KUKA KRL program: EPS_2_25252_PD2_A_20250919023702.src

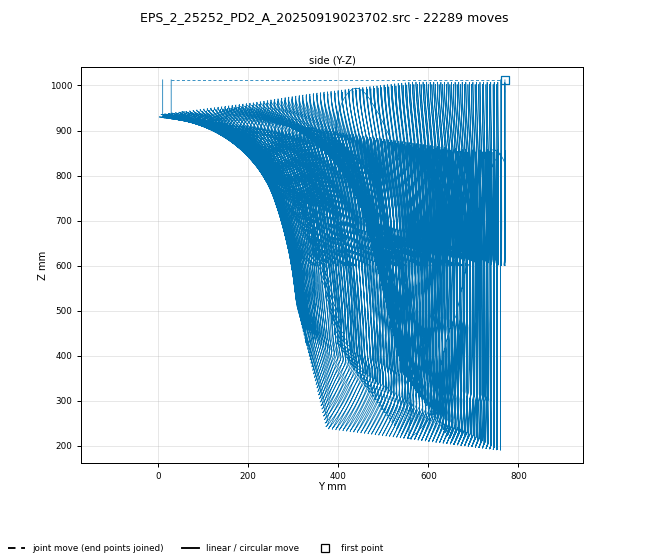
[picture p0: tool path of EPS_2_25252_PD2_A_20250919023702.src, 22289 of 22291 moves have a stored position in this frame; points joined in program order, loops and branches not executed]
&ACCESS RVP
&REL 4
&COMMENT QRS 19112012
&PARAM EDITMASK = *
DEF PART()
EXT BAS (BAS_COMMAND :IN,REAL :IN )
INT I
BAS (#INITMOV,0 )

;KUKA QRS Post kuka4.cps  Date:22-06-2017 !

File_ID=2839

QRS_PRE_INIT()

;Init var - Until changes are made in qrs_pre_init
Outlet_Square_prg=0
Inlet_1_Square_prg=0
Inlet_2_Square_prg=0
Inlet_3_Square_prg=0
Inlet_4_Square_prg=0
Inlet_5_Square_prg=0

Outlet_1={X 0.000, Y 562.000, Z 659.500, B 0.000, E1 0.000 }
Outlet_1={X 0.000, Y 562.000, Z 659.500, B 0.000, E1 0.000 }
Inlet_1={X 0.000, Y 675.710, Z 469.500, B 0.000, E1 90.000 }
Inlet_2={X 0.000, Y 612.000, Z 586.000, B 0.000, E1 180.000 }
Inlet_1={X 0.000, Y 675.710, Z 469.500, B 0.000, E1 90.000 }
Inlet_2={X 0.000, Y 612.000, Z 586.000, B 0.000, E1 180.000 }
Outlet_1_type=686
Inlet_1_type=366
Inlet_2_type=533
Inlet_1_type=366
Inlet_2_type=533
;QRS#1=Sidecore dimensions
;QRS#2=675-27" Concrete
;QRS#3=375-15" PVC SDR 35
;QRS#4=525-21" Concrete
;QRS#5=
;QRS#6=
;QRS#7=
;QRS#8=
;QRS#9=S306-38L
;QRS#10=20Y PSX
;QRS#11=S306-32
;QRS#12=
;QRS#13=
;QRS#14=
;QRS#15=
;QRS#16=1524x152x1448 4,75'
;QRS#17=EPS Height
;QRS#18=1002,5
;QRS#19=*
;QRS#20= UPDATED VERSION 22-06-2017
;QRS#21=*
Outlet_Square=0550
Inlet_1_Square=0250
Inlet_2_Square=0350
Inlet_3_Square=0
Inlet_4_Square=0
Inlet_5_Square=0
Mill_Square=1
Outlet_Square_Prg=265
Inlet_1_Square_prg=252
Inlet_2_Square_prg=263
Inlet_1_Square_prg=252
Inlet_2_Square_prg=263

QRS_INIT()

$ADVANCE=5

; T1
PTP {E1 171.717,E2 171.717}
PTP {X 0,Y 769.965,A -85,B 0,C 180,E1 171.717,E2 171.717,E3 0,E4 0,E5 0,E6 0}
QRS_SPEED_INIT()
LIN {X 0,Y 769.965,Z 1012.5,A -85,B 0,C 180,E1 171.717,E2 171.717,E3 0,E4 0,E5 0,E6 0} C_VEL
LIN {X 0,Y 769.965,Z 837.821,A -85,B 0,C 180,E1 171.717,E2 171.717} C_VEL
LIN {X 0,Y 769.965,Z 829.438,A -85,B 0,C 180,E1 171.717,E2 171.717} C_VEL
LIN {X 0,Y 769.933,Z 827.68,A -85,B 0,C 180,E1 171.937,E2 171.937} C_VEL
LIN {X 0,Y 769.905,Z 832.409,A -85,B 0,C 180,E1 172.585,E2 172.585} C_VEL
LIN {X 0,Y 769.947,Z 836.302,A -85,B 0,C 180,E1 173.179,E2 173.179} C_VEL
LIN {X 0,Y 769.972,Z 840.225,A -85,B 0,C 180,E1 173.851,E2 173.851} C_VEL
LIN {X 0,Y 769.915,Z 844.055,A -85,B 0,C 180,E1 174.598,E2 174.598} C_VEL
LIN {X 0,Y 769.912,Z 845.802,A -85,B 0,C 180,E1 174.971,E2 174.971} C_VEL
LIN {X 0,Y 769.959,Z 848.792,A -85,B 0,C 180,E1 175.718,E2 175.718} C_VEL
LIN {X 0,Y 769.933,Z 851.274,A -85,B 0,C 180,E1 176.464,E2 176.464} C_VEL
LIN {X 0,Y 769.879,Z 853.258,A -85,B 0,C 180,E1 177.209,E2 177.209} C_VEL
LIN {X 0,Y 769.914,Z 854.732,A -85,B 0,C 180,E1 177.954,E2 177.954} C_VEL
LIN {X 0,Y 769.942,Z 856.064,A -85,B 0,C 180,E1 179.07,E2 179.07} C_VEL
LIN {X 0,Y 769.898,Z 856.296,A -85,B 0,C 180,E1 179.442,E2 179.442} C_VEL
LIN {X 0,Y 769.889,Z 856.381,A -85,B 0,C 180,E1 180.186,E2 180.186} C_VEL
LIN {X 0,Y 769.977,Z 855.974,A -85,B 0,C 180,E1 180.93,E2 180.93} C_VEL
LIN {X 0,Y 769.909,Z 854.599,A -85,B 0,C 180,E1 182.046,E2 182.046} C_VEL
LIN {X 0,Y 769.9,Z 853.054,A -85,B 0,C 180,E1 182.791,E2 182.791} C_VEL
LIN {X 0,Y 769.972,Z 850.99,A -85,B 0,C 180,E1 183.536,E2 183.536} C_VEL
LIN {X 0,Y 769.944,Z 848.445,A -85,B 0,C 180,E1 184.282,E2 184.282} C_VEL
LIN {X 0,Y 769.922,Z 845.378,A -85,B 0,C 180,E1 185.028,E2 185.028} C_VEL
LIN {X 0,Y 769.979,Z 841.746,A -85,B 0,C 180,E1 185.775,E2 185.775} C_VEL
LIN {X 0,Y 769.972,Z 837.553,A -85,B 0,C 180,E1 186.524,E2 186.524} C_VEL
LIN {X 0,Y 769.927,Z 832.231,A -85,B 0,C 180,E1 187.35,E2 187.35} C_VEL
LIN {X 0,Y 769.956,Z 827.402,A -85,B 0,C 180,E1 188.009,E2 188.009} C_VEL
LIN {X 0,Y 769.993,Z 820.295,A -85,B 0,C 180,E1 188.87,E2 188.87} C_VEL
LIN {X 0,Y 769.952,Z 813.615,A -85,B 0,C 180,E1 189.577,E2 189.577} C_VEL
LIN {X 0,Y 769.982,Z 807.441,A -85,B 0,C 180,E1 190.166,E2 190.166} C_VEL
LIN {X 0,Y 770.001,Z 800.638,A -85,B 0,C 180,E1 190.757,E2 190.757} C_VEL
LIN {X 0,Y 769.976,Z 793.13,A -85,B 0,C 180,E1 191.35,E2 191.35} C_VEL
LIN {X 0,Y 769.977,Z 786.516,A -85,B 0,C 180,E1 191.824,E2 191.824} C_VEL
LIN {X 0,Y 770.007,Z 779.283,A -85,B 0,C 180,E1 192.299,E2 192.299} C_VEL
LIN {X 0,Y 770.028,Z 770.311,A -85,B 0,C 180,E1 192.835,E2 192.835} C_VEL
LIN {X 0,Y 770.01,Z 760.228,A -85,B 0,C 180,E1 193.372,E2 193.372} C_VEL
LIN {X 0,Y 769.98,Z 749.957,A -85,B 0,C 180,E1 193.851,E2 193.851} C_VEL
LIN {X 0,Y 770.013,Z 741.446,A -85,B 0,C 180,E1 194.205,E2 194.205} C_VEL
LIN {X 0,Y 770.034,Z 733.818,A -85,B 0,C 180,E1 194.492,E2 194.492} C_VEL
LIN {X 0,Y 770.019,Z 725.132,A -85,B 0,C 180,E1 194.785,E2 194.785} C_VEL
LIN {X 0,Y 770.006,Z 716.933,A -85,B 0,C 180,E1 195.031,E2 195.031} C_VEL
LIN {X 0,Y 770.046,Z 705.499,A -85,B 0,C 180,E1 195.319,E2 195.319} C_VEL
LIN {X 0,Y 770.032,Z 695.572,A -85,B 0,C 180,E1 195.528,E2 195.528} C_VEL
LIN {X 0,Y 769.952,Z 685.922,A -85,B 0,C 180,E1 195.696,E2 195.696} C_VEL
LIN {X 0,Y 769.969,Z 676.893,A -85,B 0,C 180,E1 195.819,E2 195.819} C_VEL
LIN {X 0,Y 769.906,Z 653.796,A -85,B 0,C 180,E1 196.051,E2 196.051} C_VEL
LIN {X 0,Y 769.714,Z 601.31,A -85,B 0,C 180,E1 196.558,E2 196.558} C_VEL
LIN {X 0,Y 769.999,Z 601.31,A -85,B 0,C 180,E1 196.75,E2 196.75} C_VEL
LIN {X 0,Y 769.993,Z 601.31,A -85,B 0,C 180,E1 199.928,E2 199.928} C_VEL
LIN {X 0,Y 769.932,Z 601.31,A -85,B 0,C 180,E1 203.94,E2 203.94} C_VEL
LIN {X 0,Y 769.57,Z 601.31,A -85,B 0,C 180,E1 206.729,E2 206.729} C_VEL
LIN {X 0,Y 769.926,Z 601.31,A -85,B 0,C 180,E1 208.081,E2 208.081} C_VEL
LIN {X 0,Y 769.514,Z 601.31,A -85,B 0,C 180,E1 210.601,E2 210.601} C_VEL
LIN {X 0,Y 769.889,Z 601.31,A -85,B 0,C 180,E1 212.389,E2 212.389} C_VEL
LIN {X 0,Y 769.475,Z 601.31,A -85,B 0,C 180,E1 214.641,E2 214.641} C_VEL
LIN {X 0,Y 770.073,Z 601.31,A -85,B 0,C 180,E1 217.326,E2 217.326} C_VEL
LIN {X 0,Y 769.817,Z 601.31,A -85,B 0,C 180,E1 221.727,E2 221.727} C_VEL
LIN {X 0,Y 769.873,Z 601.31,A -85,B 0,C 180,E1 223.074,E2 223.074} C_VEL
LIN {X 0,Y 769.861,Z 601.31,A -85,B 0,C 180,E1 224.268,E2 224.268} C_VEL
LIN {X 0,Y 769.772,Z 601.31,A -85,B 0,C 180,E1 225.726,E2 225.726} C_VEL
LIN {X 0,Y 769.765,Z 601.31,A -85,B 0,C 180,E1 229.733,E2 229.733} C_VEL
LIN {X 0,Y 769.804,Z 601.31,A -85,B 0,C 180,E1 230.718,E2 230.718} C_VEL
LIN {X 0,Y 769.413,Z 601.31,A -85,B 0,C 180,E1 233.061,E2 233.061} C_VEL
LIN {X 0,Y 769.839,Z 601.31,A -85,B 0,C 180,E1 235.377,E2 235.377} C_VEL
LIN {X 0,Y 770.07,Z 601.31,A -85,B 0,C 180,E1 240.027,E2 240.027} C_VEL
LIN {X 0,Y 769.183,Z 601.31,A -85,B 0,C 180,E1 240.219,E2 240.219} C_VEL
LIN {X 0,Y 767.602,Z 601.31,A -85,B 0,C 180,E1 240.325,E2 240.325} C_VEL
LIN {X 0,Y 769.564,Z 617.584,A -85,B 0,C 180,E1 240.592,E2 240.592} C_VEL
LIN {X 0,Y 769.685,Z 674.251,A -85,B 0,C 180,E1 241.19,E2 241.19} C_VEL
LIN {X 0,Y 769.843,Z 693.525,A -85,B 0,C 180,E1 241.423,E2 241.423} C_VEL
LIN {X 0,Y 769.775,Z 704.388,A -85,B 0,C 180,E1 241.585,E2 241.585} C_VEL
LIN {X 0,Y 769.63,Z 714.271,A -85,B 0,C 180,E1 241.743,E2 241.743} C_VEL
LIN {X 0,Y 769.801,Z 732.539,A -85,B 0,C 180,E1 242.131,E2 242.131} C_VEL
LIN {X 0,Y 769.675,Z 749.053,A -85,B 0,C 180,E1 242.539,E2 242.539} C_VEL
LIN {X 0,Y 769.872,Z 765.18,A -85,B 0,C 180,E1 243.017,E2 243.017} C_VEL
LIN {X 0,Y 769.857,Z 781.112,A -85,B 0,C 180,E1 243.548,E2 243.548} C_VEL
LIN {X 0,Y 769.803,Z 791.905,A -85,B 0,C 180,E1 243.946,E2 243.946} C_VEL
LIN {X 0,Y 769.91,Z 806.611,A -85,B 0,C 180,E1 244.549,E2 244.549} C_VEL
LIN {X 0,Y 769.911,Z 814.435,A -85,B 0,C 180,E1 244.896,E2 244.896} C_VEL
LIN {X 0,Y 769.862,Z 826.837,A -85,B 0,C 180,E1 245.477,E2 245.477} C_VEL
LIN {X 0,Y 769.906,Z 840.576,A -85,B 0,C 180,E1 246.186,E2 246.186} C_VEL
LIN {X 0,Y 769.93,Z 854.071,A -85,B 0,C 180,E1 246.947,E2 246.947} C_VEL
LIN {X 0,Y 769.916,Z 866.978,A -85,B 0,C 180,E1 247.739,E2 247.739} C_VEL
LIN {X 0,Y 769.895,Z 879.836,A -85,B 0,C 180,E1 248.599,E2 248.599} C_VEL
LIN {X 0,Y 769.945,Z 891.695,A -85,B 0,C 180,E1 249.463,E2 249.463} C_VEL
LIN {X 0,Y 769.92,Z 904.013,A -85,B 0,C 180,E1 250.441,E2 250.441} C_VEL
LIN {X 0,Y 769.891,Z 914.05,A -85,B 0,C 180,E1 251.301,E2 251.301} C_VEL
LIN {X 0,Y 769.981,Z 925.132,A -85,B 0,C 180,E1 252.343,E2 252.343} C_VEL
LIN {X 0,Y 769.835,Z 934.509,A -85,B 0,C 180,E1 253.29,E2 253.29} C_VEL
LIN {X 0,Y 769.849,Z 944.258,A -85,B 0,C 180,E1 254.375,E2 254.375} C_VEL
LIN {X 0,Y 769.965,Z 953.171,A -85,B 0,C 180,E1 255.469,E2 255.469} C_VEL
LIN {X 0,Y 769.771,Z 961.783,A -85,B 0,C 180,E1 256.624,E2 256.624} C_VEL
LIN {X 0,Y 769.79,Z 968.235,A -85,B 0,C 180,E1 257.578,E2 257.578} C_VEL
LIN {X 0,Y 769.967,Z 975.408,A -85,B 0,C 180,E1 258.769,E2 258.769} C_VEL
LIN {X 0,Y 769.797,Z 981.796,A -85,B 0,C 180,E1 259.949,E2 259.949} C_VEL
LIN {X 0,Y 769.926,Z 988.323,A -85,B 0,C 180,E1 261.365,E2 261.365} C_VEL
LIN {X 0,Y 769.906,Z 991.578,A -85,B 0,C 180,E1 262.177,E2 262.177} C_VEL
LIN {X 0,Y 769.774,Z 994.107,A -85,B 0,C 180,E1 262.86,E2 262.86} C_VEL
LIN {X 0,Y 769.774,Z 997.359,A -85,B 0,C 180,E1 263.849,E2 263.849} C_VEL
LIN {X 0,Y 769.873,Z 999.367,A -85,B 0,C 180,E1 264.598,E2 264.598} C_VEL
LIN {X 0,Y 769.914,Z 1001.173,A -85,B 0,C 180,E1 265.345,E2 265.345} C_VEL
LIN {X 0,Y 769.719,Z 1003.452,A -85,B 0,C 180,E1 266.463,E2 266.463} C_VEL
LIN {X 0,Y 769.72,Z 1004.562,A -85,B 0,C 180,E1 267.208,E2 267.208} C_VEL
LIN {X 0,Y 769.916,Z 1005.682,A -85,B 0,C 180,E1 268.326,E2 268.326} C_VEL
LIN {X 0,Y 769.876,Z 1006.173,A -85,B 0,C 180,E1 269.07,E2 269.07} C_VEL
LIN {X 0,Y 769.751,Z 1006.206,A -85,B 0,C 180,E1 270.93,E2 270.93} C_VEL
LIN {X 0,Y 769.984,Z 1005.332,A -85,B 0,C 180,E1 272.046,E2 272.046} C_VEL
LIN {X 0,Y 769.855,Z 1004.527,A -85,B 0,C 180,E1 272.791,E2 272.791} C_VEL
LIN {X 0,Y 769.749,Z 1002.792,A -85,B 0,C 180,E1 273.91,E2 273.91} C_VEL
LIN {X 0,Y 769.834,Z 1001.194,A -85,B 0,C 180,E1 274.656,E2 274.656} C_VEL
LIN {X 0,Y 769.978,Z 999.341,A -85,B 0,C 180,E1 275.401,E2 275.401} C_VEL
LIN {X 0,Y 769.818,Z 997.349,A -85,B 0,C 180,E1 276.151,E2 276.151} C_VEL
LIN {X 0,Y 769.74,Z 993.279,A -85,B 0,C 180,E1 277.39,E2 277.39} C_VEL
LIN {X 0,Y 769.934,Z 987.309,A -85,B 0,C 180,E1 278.87,E2 278.87} C_VEL
LIN {X 0,Y 769.785,Z 981.8,A -85,B 0,C 180,E1 280.051,E2 280.051} C_VEL
LIN {X 0,Y 769.877,Z 975.429,A -85,B 0,C 180,E1 281.232,E2 281.232} C_VEL
LIN {X 0,Y 769.921,Z 969.675,A -85,B 0,C 180,E1 282.181,E2 282.181} C_VEL
LIN {X 0,Y 769.807,Z 965.001,A -85,B 0,C 180,E1 282.898,E2 282.898} C_VEL
LIN {X 0,Y 769.804,Z 960.105,A -85,B 0,C 180,E1 283.615,E2 283.615} C_VEL
LIN {X 0,Y 769.984,Z 950.904,A -85,B 0,C 180,E1 284.816,E2 284.816} C_VEL
LIN {X 0,Y 769.84,Z 942.603,A -85,B 0,C 180,E1 285.819,E2 285.819} C_VEL
LIN {X 0,Y 769.822,Z 932.765,A -85,B 0,C 180,E1 286.895,E2 286.895} C_VEL
LIN {X 0,Y 769.968,Z 921.995,A -85,B 0,C 180,E1 287.962,E2 287.962} C_VEL
LIN {X 0,Y 769.882,Z 911.261,A -85,B 0,C 180,E1 288.944,E2 288.944} C_VEL
LIN {X 0,Y 769.912,Z 901.04,A -85,B 0,C 180,E1 289.806,E2 289.806} C_VEL
LIN {X 0,Y 769.957,Z 889.67,A -85,B 0,C 180,E1 290.689,E2 290.689} C_VEL
LIN {X 0,Y 769.903,Z 877.271,A -85,B 0,C 180,E1 291.578,E2 291.578} C_VEL
LIN {X 0,Y 769.914,Z 864.609,A -85,B 0,C 180,E1 292.411,E2 292.411} C_VEL
LIN {X 0,Y 769.919,Z 850.802,A -85,B 0,C 180,E1 293.243,E2 293.243} C_VEL
LIN {X 0,Y 769.908,Z 836.618,A -85,B 0,C 180,E1 294.024,E2 294.024} C_VEL
LIN {X 0,Y 769.845,Z 823.461,A -85,B 0,C 180,E1 294.69,E2 294.69} C_VEL
LIN {X 0,Y 769.907,Z 808.968,A -85,B 0,C 180,E1 295.353,E2 295.353} C_VEL
LIN {X 0,Y 769.866,Z 792.045,A -85,B 0,C 180,E1 296.046,E2 296.046} C_VEL
LIN {X 0,Y 769.796,Z 779.364,A -85,B 0,C 180,E1 296.519,E2 296.519} C_VEL
LIN {X 0,Y 769.896,Z 761.332,A -85,B 0,C 180,E1 297.102,E2 297.102} C_VEL
LIN {X 0,Y 769.784,Z 744.594,A -85,B 0,C 180,E1 297.576,E2 297.576} C_VEL
LIN {X 0,Y 769.706,Z 735.342,A -85,B 0,C 180,E1 297.804,E2 297.804} C_VEL
LIN {X 0,Y 769.828,Z 726.233,A -85,B 0,C 180,E1 298.006,E2 298.006} C_VEL
LIN {X 0,Y 769.852,Z 711.957,A -85,B 0,C 180,E1 298.289,E2 298.289} C_VEL
LIN {X 0,Y 769.605,Z 695.19,A -85,B 0,C 180,E1 298.566,E2 298.566} C_VEL
LIN {X 0,Y 769.681,Z 674.237,A -85,B 0,C 180,E1 298.811,E2 298.811} C_VEL
LIN {X 0,Y 769.572,Z 617.494,A -85,B 0,C 180,E1 299.409,E2 299.409} C_VEL
LIN {X 0,Y 769.452,Z 601.31,A -85,B 0,C 180,E1 299.814,E2 299.814} C_VEL
LIN {X 0,Y 770.022,Z 601.31,A -85,B 0,C 180,E1 300.206,E2 300.206} C_VEL
LIN {X 0,Y 769.962,Z 601.31,A -85,B 0,C 180,E1 302.385,E2 302.385} C_VEL
LIN {X 0,Y 769.449,Z 601.31,A -85,B 0,C 180,E1 304.642,E2 304.642} C_VEL
LIN {X 0,Y 770.005,Z 601.31,A -85,B 0,C 180,E1 307.32,E2 307.32} C_VEL
LIN {X 0,Y 769.808,Z 601.31,A -85,B 0,C 180,E1 311.728,E2 311.728} C_VEL
LIN {X 0,Y 769.854,Z 601.31,A -85,B 0,C 180,E1 313.073,E2 313.073} C_VEL
LIN {X 0,Y 769.83,Z 601.31,A -85,B 0,C 180,E1 314.27,E2 314.27} C_VEL
LIN {X 0,Y 769.731,Z 601.31,A -85,B 0,C 180,E1 315.723,E2 315.723} C_VEL
LIN {X 0,Y 769.801,Z 601.31,A -85,B 0,C 180,E1 319.73,E2 319.73} C_VEL
LIN {X 0,Y 769.843,Z 601.31,A -85,B 0,C 180,E1 320.721,E2 320.721} C_VEL
LIN {X 0,Y 769.435,Z 601.31,A -85,B 0,C 180,E1 323.062,E2 323.062} C_VEL
LIN {X 0,Y 769.851,Z 601.31,A -85,B 0,C 180,E1 325.378,E2 325.378} C_VEL
LIN {X 0,Y 769.987,Z 601.31,A -85,B 0,C 180,E1 329.339,E2 329.339} C_VEL
LIN {X 0,Y 769.827,Z 601.31,A -85,B 0,C 180,E1 333.233,E2 333.233} C_VEL
LIN {X 0,Y 769.918,Z 601.31,A -85,B 0,C 180,E1 334.007,E2 334.007} C_VEL
LIN {X 0,Y 769.986,Z 601.31,A -85,B 0,C 180,E1 337.687,E2 337.687} C_VEL
LIN {X 0,Y 769.954,Z 601.31,A -85,B 0,C 180,E1 338.08,E2 338.08} C_VEL
LIN {X 0,Y 769.968,Z 601.31,A -85,B 0,C 180,E1 342.038,E2 342.038} C_VEL
LIN {X 0,Y 769.699,Z 601.31,A -85,B 0,C 180,E1 343.977,E2 343.977} C_VEL
LIN {X 0,Y 769.8,Z 601.31,A -85,B 0,C 180,E1 345.906,E2 345.906} C_VEL
LIN {X 0,Y 769.997,Z 601.31,A -85,B 0,C 180,E1 349.716,E2 349.716} C_VEL
LIN {X 0,Y 770.018,Z 601.31,A -85,B 0,C 180,E1 353.477,E2 353.477} C_VEL
LIN {X 0,Y 770.056,Z 601.31,A -85,B 0,C 180,E1 357.209,E2 357.209} C_VEL
LIN {X 0,Y 770.07,Z 601.31,A -85,B 0,C 180,E1 360.93,E2 360.93} C_VEL
LIN {X 0,Y 770.058,Z 601.31,A -85,B 0,C 180,E1 364.654,E2 364.654} C_VEL
LIN {X 0,Y 770.03,Z 601.31,A -85,B 0,C 180,E1 368.399,E2 368.399} C_VEL
LIN {X 0,Y 770.008,Z 601.31,A -85,B 0,C 180,E1 372.18,E2 372.18} C_VEL
LIN {X 0,Y 769.992,Z 601.31,A -85,B 0,C 180,E1 376.016,E2 376.016} C_VEL
LIN {X 0,Y 769.858,Z 601.31,A -85,B 0,C 180,E1 376.716,E2 376.716} C_VEL
LIN {X 0,Y 769.973,Z 601.31,A -85,B 0,C 180,E1 379.928,E2 379.928} C_VEL
LIN {X 0,Y 769.599,Z 601.31,A -85,B 0,C 180,E1 382.243,E2 382.243} C_VEL
LIN {X 0,Y 769.955,Z 601.31,A -85,B 0,C 180,E1 383.94,E2 383.94} C_VEL
LIN {X 0,Y 769.585,Z 601.31,A -85,B 0,C 180,E1 386.731,E2 386.731} C_VEL
LIN {X 0,Y 769.933,Z 601.31,A -85,B 0,C 180,E1 388.08,E2 388.08} C_VEL
LIN {X 0,Y 769.518,Z 601.31,A -85,B 0,C 180,E1 390.602,E2 390.602} C_VEL
LIN {X 0,Y 769.883,Z 601.31,A -85,B 0,C 180,E1 392.389,E2 392.389} C_VEL
LIN {X 0,Y 769.467,Z 601.31,A -85,B 0,C 180,E1 394.642,E2 394.642} C_VEL
LIN {X 0,Y 770.07,Z 601.31,A -85,B 0,C 180,E1 397.327,E2 397.327} C_VEL
LIN {X 0,Y 769.807,Z 601.31,A -85,B 0,C 180,E1 401.728,E2 401.728} C_VEL
LIN {X 0,Y 769.861,Z 601.31,A -85,B 0,C 180,E1 403.074,E2 403.074} C_VEL
LIN {X 0,Y 769.847,Z 601.31,A -85,B 0,C 180,E1 404.269,E2 404.269} C_VEL
LIN {X 0,Y 769.76,Z 601.31,A -85,B 0,C 180,E1 405.725,E2 405.725} C_VEL
LIN {X 0,Y 769.806,Z 601.31,A -85,B 0,C 180,E1 409.729,E2 409.729} C_VEL
LIN {X 0,Y 769.843,Z 601.31,A -85,B 0,C 180,E1 410.721,E2 410.721} C_VEL
LIN {X 0,Y 769.432,Z 601.31,A -85,B 0,C 180,E1 413.062,E2 413.062} C_VEL
LIN {X 0,Y 769.848,Z 601.31,A -85,B 0,C 180,E1 415.378,E2 415.378} C_VEL
LIN {X 0,Y 770.026,Z 601.31,A -85,B 0,C 180,E1 419.334,E2 419.334} C_VEL
LIN {X 0,Y 769.851,Z 601.31,A -85,B 0,C 180,E1 423.23,E2 423.23} C_VEL
LIN {X 0,Y 769.959,Z 601.31,A -85,B 0,C 180,E1 424.009,E2 424.009} C_VEL
LIN {X 0,Y 769.955,Z 601.31,A -85,B 0,C 180,E1 427.045,E2 427.045} C_VEL
LIN {X 0,Y 769.914,Z 601.31,A -85,B 0,C 180,E1 427.416,E2 427.416} C_VEL
LIN {X 0,Y 769.332,Z 601.31,A -85,B 0,C 180,E1 427.512,E2 427.512} C_VEL
LIN {X 0,Y 769.77,Z 613.478,A -85,B 0,C 180,E1 427.681,E2 427.681} C_VEL
LIN {X 0,Y 769.925,Z 626.518,A -85,B 0,C 180,E1 427.898,E2 427.898} C_VEL
LIN {X 0,Y 769.9,Z 639.512,A -85,B 0,C 180,E1 428.158,E2 428.158} C_VEL
LIN {X 0,Y 769.934,Z 650.634,A -85,B 0,C 180,E1 428.42,E2 428.42} C_VEL
LIN {X 0,Y 769.971,Z 664.457,A -85,B 0,C 180,E1 428.803,E2 428.803} C_VEL
LIN {X 0,Y 769.873,Z 677.696,A -85,B 0,C 180,E1 429.223,E2 429.223} C_VEL
LIN {X 0,Y 769.961,Z 690.101,A -85,B 0,C 180,E1 429.675,E2 429.675} C_VEL
LIN {X 0,Y 769.972,Z 701.475,A -85,B 0,C 180,E1 430.134,E2 430.134} C_VEL
LIN {X 0,Y 769.967,Z 713.804,A -85,B 0,C 180,E1 430.689,E2 430.689} C_VEL
LIN {X 0,Y 769.971,Z 724.932,A -85,B 0,C 180,E1 431.242,E2 431.242} C_VEL
LIN {X 0,Y 769.975,Z 736.111,A -85,B 0,C 180,E1 431.855,E2 431.855} C_VEL
LIN {X 0,Y 769.966,Z 746.59,A -85,B 0,C 180,E1 432.485,E2 432.485} C_VEL
LIN {X 0,Y 769.946,Z 756.745,A -85,B 0,C 180,E1 433.152,E2 433.152} C_VEL
LIN {X 0,Y 769.972,Z 765.735,A -85,B 0,C 180,E1 433.794,E2 433.794} C_VEL
LIN {X 0,Y 769.97,Z 775.722,A -85,B 0,C 180,E1 434.575,E2 434.575} C_VEL
LIN {X 0,Y 769.918,Z 783.892,A -85,B 0,C 180,E1 435.268,E2 435.268} C_VEL
LIN {X 0,Y 769.953,Z 792.116,A -85,B 0,C 180,E1 436.029,E2 436.029} C_VEL
LIN {X 0,Y 769.948,Z 800.384,A -85,B 0,C 180,E1 436.866,E2 436.866} C_VEL
LIN {X 0,Y 769.869,Z 807.913,A -85,B 0,C 180,E1 437.699,E2 437.699} C_VEL
LIN {X 0,Y 769.913,Z 814.731,A -85,B 0,C 180,E1 438.531,E2 438.531} C_VEL
LIN {X 0,Y 769.977,Z 820.092,A -85,B 0,C 180,E1 439.243,E2 439.243} C_VEL
LIN {X 0,Y 769.842,Z 826.554,A -85,B 0,C 180,E1 440.186,E2 440.186} C_VEL
LIN {X 0,Y 769.864,Z 832.255,A -85,B 0,C 180,E1 441.129,E2 441.129} C_VEL
LIN {X 0,Y 769.949,Z 837.839,A -85,B 0,C 180,E1 442.193,E2 442.193} C_VEL
LIN {X 0,Y 769.808,Z 842.358,A -85,B 0,C 180,E1 443.172,E2 443.172} C_VEL
LIN {X 0,Y 769.844,Z 846.42,A -85,B 0,C 180,E1 444.224,E2 444.224} C_VEL
LIN {X 0,Y 769.974,Z 848.895,A -85,B 0,C 180,E1 444.972,E2 444.972} C_VEL
LIN {X 0,Y 769.82,Z 851.939,A -85,B 0,C 180,E1 446.091,E2 446.091} C_VEL
LIN {X 0,Y 769.844,Z 854.142,A -85,B 0,C 180,E1 447.209,E2 447.209} C_VEL
LIN {X 0,Y 769.987,Z 855.212,A -85,B 0,C 180,E1 447.954,E2 447.954} C_VEL
LIN {X 0,Y 769.798,Z 856.215,A -85,B 0,C 180,E1 449.07,E2 449.07} C_VEL
LIN {X 0,Y 769.838,Z 856.173,A -85,B 0,C 180,E1 450.93,E2 450.93} C_VEL
LIN {X 0,Y 769.984,Z 855.479,A -85,B 0,C 180,E1 451.674,E2 451.674} C_VEL
LIN {X 0,Y 769.805,Z 854.02,A -85,B 0,C 180,E1 452.792,E2 452.792} C_VEL
LIN {X 0,Y 769.819,Z 852.527,A -85,B 0,C 180,E1 453.537,E2 453.537} C_VEL
LIN {X 0,Y 769.977,Z 849.68,A -85,B 0,C 180,E1 454.655,E2 454.655} C_VEL
LIN {X 0,Y 769.889,Z 847.357,A -85,B 0,C 180,E1 455.402,E2 455.402} C_VEL
LIN {X 0,Y 769.839,Z 844.699,A -85,B 0,C 180,E1 456.151,E2 456.151} C_VEL
LIN {X 0,Y 769.885,Z 842.02,A -85,B 0,C 180,E1 456.818,E2 456.818} C_VEL
LIN {X 0,Y 769.948,Z 837.617,A -85,B 0,C 180,E1 457.765,E2 457.765} C_VEL
LIN {X 0,Y 769.837,Z 831.728,A -85,B 0,C 180,E1 458.872,E2 458.872} C_VEL
LIN {X 0,Y 769.928,Z 825.932,A -85,B 0,C 180,E1 459.813,E2 459.813} C_VEL
LIN {X 0,Y 769.96,Z 819.413,A -85,B 0,C 180,E1 460.758,E2 460.758} C_VEL
LIN {X 0,Y 769.873,Z 812.124,A -85,B 0,C 180,E1 461.707,E2 461.707} C_VEL
LIN {X 0,Y 769.932,Z 805.037,A -85,B 0,C 180,E1 462.539,E2 462.539} C_VEL
LIN {X 0,Y 769.955,Z 797.229,A -85,B 0,C 180,E1 463.373,E2 463.373} C_VEL
LIN {X 0,Y 769.901,Z 789.949,A -85,B 0,C 180,E1 464.092,E2 464.092} C_VEL
LIN {X 0,Y 769.937,Z 780.882,A -85,B 0,C 180,E1 464.905,E2 464.905} C_VEL
LIN {X 0,Y 769.975,Z 772.306,A -85,B 0,C 180,E1 465.611,E2 465.611} C_VEL
LIN {X 0,Y 769.956,Z 763.175,A -85,B 0,C 180,E1 466.305,E2 466.305} C_VEL
LIN {X 0,Y 769.981,Z 753.102,A -85,B 0,C 180,E1 467.004,E2 467.004} C_VEL
LIN {X 0,Y 769.987,Z 742.67,A -85,B 0,C 180,E1 467.666,E2 467.666} C_VEL
LIN {X 0,Y 769.967,Z 732.34,A -85,B 0,C 180,E1 468.268,E2 468.268} C_VEL
LIN {X 0,Y 769.962,Z 721.993,A -85,B 0,C 180,E1 468.82,E2 468.82} C_VEL
LIN {X 0,Y 769.922,Z 710.569,A -85,B 0,C 180,E1 469.374,E2 469.374} C_VEL
LIN {X 0,Y 769.975,Z 697.801,A -85,B 0,C 180,E1 469.928,E2 469.928} C_VEL
LIN {X 0,Y 769.954,Z 685.56,A -85,B 0,C 180,E1 470.406,E2 470.406} C_VEL
LIN {X 0,Y 769.89,Z 673.731,A -85,B 0,C 180,E1 470.819,E2 470.819} C_VEL
LIN {X 0,Y 769.972,Z 661.358,A -85,B 0,C 180,E1 471.197,E2 471.197} C_VEL
LIN {X 0,Y 769.929,Z 647.309,A -85,B 0,C 180,E1 471.57,E2 471.57} C_VEL
LIN {X 0,Y 769.899,Z 636.718,A -85,B 0,C 180,E1 471.815,E2 471.815} C_VEL
LIN {X 0,Y 769.944,Z 621.218,A -85,B 0,C 180,E1 472.104,E2 472.104} C_VEL
LIN {X 0,Y 769.757,Z 607.881,A -85,B 0,C 180,E1 472.307,E2 472.307} C_VEL
LIN {X 0,Y 768.741,Z 601.482,A -85,B 0,C 180,E1 472.413,E2 472.413} C_VEL
LIN {X 0,Y 768.776,Z 601.31,A -85,B 0,C 180,E1 472.422,E2 472.422} C_VEL
LIN {X 0,Y 769.387,Z 601.31,A -85,B 0,C 180,E1 472.48,E2 472.48} C_VEL
LIN {X 0,Y 770.077,Z 601.31,A -85,B 0,C 180,E1 472.757,E2 472.757} C_VEL
LIN {X 0,Y 769.92,Z 601.31,A -85,B 0,C 180,E1 473.459,E2 473.459} C_VEL
LIN {X 0,Y 769.909,Z 601.31,A -85,B 0,C 180,E1 478.081,E2 478.081} C_VEL
LIN {X 0,Y 769.513,Z 601.31,A -85,B 0,C 180,E1 480.601,E2 480.601} C_VEL
LIN {X 0,Y 769.893,Z 601.31,A -85,B 0,C 180,E1 482.389,E2 482.389} C_VEL
LIN {X 0,Y 769.547,Z 601.31,A -85,B 0,C 180,E1 484.084,E2 484.084} C_VEL
LIN {X 0,Y 769.998,Z 601.31,A -85,B 0,C 180,E1 487.319,E2 487.319} C_VEL
LIN {X 0,Y 769.807,Z 601.31,A -85,B 0,C 180,E1 491.728,E2 491.728} C_VEL
LIN {X 0,Y 769.878,Z 601.31,A -85,B 0,C 180,E1 493.075,E2 493.075} C_VEL
LIN {X 0,Y 769.861,Z 601.31,A -85,B 0,C 180,E1 494.268,E2 494.268} C_VEL
LIN {X 0,Y 769.782,Z 601.31,A -85,B 0,C 180,E1 495.726,E2 495.726} C_VEL
LIN {X 0,Y 769.798,Z 601.31,A -85,B 0,C 180,E1 499.73,E2 499.73} C_VEL
LIN {X 0,Y 769.828,Z 601.31,A -85,B 0,C 180,E1 500.72,E2 500.72} C_VEL
LIN {X 0,Y 769.429,Z 601.31,A -85,B 0,C 180,E1 503.062,E2 503.062} C_VEL
LIN {X 0,Y 769.869,Z 601.31,A -85,B 0,C 180,E1 505.379,E2 505.379} C_VEL
LIN {X 0,Y 770.008,Z 601.31,A -85,B 0,C 180,E1 509.337,E2 509.337} C_VEL
LIN {X 0,Y 769.841,Z 601.31,A -85,B 0,C 180,E1 513.231,E2 513.231} C_VEL
LIN {X 0,Y 769.933,Z 601.31,A -85,B 0,C 180,E1 514.008,E2 514.008} C_VEL
LIN {X 0,Y 769.975,Z 601.31,A -85,B 0,C 180,E1 517.689,E2 517.689} C_VEL
LIN {X 0,Y 769.897,Z 601.31,A -85,B 0,C 180,E1 518.078,E2 518.078} C_VEL
LIN {X 0,Y 770.06,Z 601.31,A -85,B 0,C 180,E1 523.067,E2 523.067} C_VEL
LIN {X 0,Y 769.734,Z 601.31,A -85,B 0,C 180,E1 523.216,E2 523.216} C_VEL
LIN {X 0,Y 768.796,Z 601.331,A -85,B 0,C 180,E1 523.334,E2 523.334} C_VEL
LIN {X 0,Y 769.689,Z 604.876,A -85,B 0,C 180,E1 523.388,E2 523.388} C_VEL
LIN {X 0,Y 769.872,Z 607.539,A -85,B 0,C 180,E1 523.418,E2 523.418} C_VEL
LIN {X 0,Y 769.92,Z 674.992,A -85,B 0,C 180,E1 524.068,E2 524.068} C_VEL
LIN {X 0,Y 769.982,Z 683.617,A -85,B 0,C 180,E1 524.18,E2 524.18} C_VEL
LIN {X 0,Y 769.998,Z 693.035,A -85,B 0,C 180,E1 524.334,E2 524.334} C_VEL
LIN {X 0,Y 769.978,Z 701.71,A -85,B 0,C 180,E1 524.505,E2 524.505} C_VEL
LIN {X 0,Y 770.04,Z 710.854,A -85,B 0,C 180,E1 524.721,E2 524.721} C_VEL
LIN {X 0,Y 770.045,Z 719.833,A -85,B 0,C 180,E1 524.966,E2 524.966} C_VEL
LIN {X 0,Y 770.015,Z 729.182,A -85,B 0,C 180,E1 525.258,E2 525.258} C_VEL
LIN {X 0,Y 769.994,Z 737.442,A -85,B 0,C 180,E1 525.55,E2 525.55} C_VEL
LIN {X 0,Y 769.997,Z 746.488,A -85,B 0,C 180,E1 525.91,E2 525.91} C_VEL
LIN {X 0,Y 770.01,Z 754.606,A -85,B 0,C 180,E1 526.269,E2 526.269} C_VEL
LIN {X 0,Y 770.022,Z 763.123,A -85,B 0,C 180,E1 526.688,E2 526.688} C_VEL
LIN {X 0,Y 770.028,Z 770.835,A -85,B 0,C 180,E1 527.106,E2 527.106} C_VEL
LIN {X 0,Y 769.994,Z 778.828,A -85,B 0,C 180,E1 527.582,E2 527.582} C_VEL
LIN {X 0,Y 770.001,Z 786.095,A -85,B 0,C 180,E1 528.057,E2 528.057} C_VEL
LIN {X 0,Y 770.001,Z 792.746,A -85,B 0,C 180,E1 528.532,E2 528.532} C_VEL
LIN {X 0,Y 770.007,Z 798.854,A -85,B 0,C 180,E1 529.006,E2 529.006} C_VEL
LIN {X 0,Y 769.999,Z 804.493,A -85,B 0,C 180,E1 529.479,E2 529.479} C_VEL
LIN {X 0,Y 769.952,Z 810.928,A -85,B 0,C 180,E1 530.069,E2 530.069} C_VEL
LIN {X 0,Y 769.954,Z 816.768,A -85,B 0,C 180,E1 530.659,E2 530.659} C_VEL
LIN {X 0,Y 769.993,Z 821.08,A -85,B 0,C 180,E1 531.13,E2 531.13} C_VEL
LIN {X 0,Y 769.937,Z 827.056,A -85,B 0,C 180,E1 531.855,E2 531.855} C_VEL
LIN {X 0,Y 769.933,Z 827.68,A -85,B 0,C 180,E1 531.937,E2 531.937} C_VEL
LIN {X 0,Y 766.018,Z 836.423,A -85,B 0,C 180,E1 533.052,E2 533.052} C_VEL
LIN {X 0,Y 762.134,Z 843.351,A -85,B 0,C 180,E1 534.211,E2 534.211} C_VEL
LIN {X 0,Y 762.11,Z 852.693,A -85,B 0,C 180,E1 536.583,E2 536.583} C_VEL
LIN {X 0,Y 762.107,Z 856.956,A -85,B 0,C 180,E1 538.862,E2 538.862} C_VEL
LIN {X 0,Y 762.133,Z 856.874,A -85,B 0,C 180,E1 541.14,E2 541.14} C_VEL
LIN {X 0,Y 762.145,Z 852.441,A -85,B 0,C 180,E1 543.42,E2 543.42} C_VEL
LIN {X 0,Y 762.16,Z 841.708,A -85,B 0,C 180,E1 546.007,E2 546.007} C_VEL
LIN {X 0,Y 762.16,Z 825.433,A -85,B 0,C 180,E1 548.431,E2 548.431} C_VEL
LIN {X 0,Y 762.225,Z 804.371,A -85,B 0,C 180,E1 550.595,E2 550.595} C_VEL
LIN {X 0,Y 762.264,Z 778.717,A -85,B 0,C 180,E1 552.483,E2 552.483} C_VEL
LIN {X 0,Y 762.285,Z 749.574,A -85,B 0,C 180,E1 554.018,E2 554.018} C_VEL
LIN {X 0,Y 762.364,Z 716.713,A -85,B 0,C 180,E1 555.193,E2 555.193} C_VEL
LIN {X 0,Y 762.384,Z 683.449,A -85,B 0,C 180,E1 555.894,E2 555.894} C_VEL
LIN {X 0,Y 762.032,Z 601.31,A -85,B 0,C 180,E1 556.733,E2 556.733} C_VEL
LIN {X 0,Y 761.727,Z 601.31,A -85,B 0,C 180,E1 560.977,E2 560.977} C_VEL
LIN {X 0,Y 761.762,Z 601.31,A -85,B 0,C 180,E1 564.686,E2 564.686} C_VEL
LIN {X 0,Y 761.732,Z 601.31,A -85,B 0,C 180,E1 568.934,E2 568.934} C_VEL
LIN {X 0,Y 761.696,Z 601.31,A -85,B 0,C 180,E1 573.339,E2 573.339} C_VEL
LIN {X 0,Y 761.844,Z 601.31,A -85,B 0,C 180,E1 578.057,E2 578.057} C_VEL
LIN {X 0,Y 761.932,Z 601.31,A -85,B 0,C 180,E1 582.63,E2 582.63} C_VEL
LIN {X 0,Y 761.799,Z 601.31,A -85,B 0,C 180,E1 585.886,E2 585.886} C_VEL
LIN {X 0,Y 761.852,Z 601.31,A -85,B 0,C 180,E1 590.851,E2 590.851} C_VEL
LIN {X 0,Y 761.649,Z 601.31,A -85,B 0,C 180,E1 596.154,E2 596.154} C_VEL
LIN {X 0,Y 762.088,Z 601.31,A -85,B 0,C 180,E1 599.869,E2 599.869} C_VEL
LIN {X 0,Y 760.847,Z 601.31,A -85,B 0,C 180,E1 600.021,E2 600.021} C_VEL
LIN {X 0,Y 762.7,Z 626.531,A -85,B 0,C 180,E1 600.396,E2 600.396} C_VEL
LIN {X 0,Y 762.797,Z 706.612,A -85,B 0,C 180,E1 601.337,E2 601.337} C_VEL
LIN {X 0,Y 762.597,Z 749.995,A -85,B 0,C 180,E1 602.29,E2 602.29} C_VEL
LIN {X 0,Y 762.592,Z 793.835,A -85,B 0,C 180,E1 603.753,E2 603.753} C_VEL
LIN {X 0,Y 762.498,Z 837.494,A -85,B 0,C 180,E1 605.773,E2 605.773} C_VEL
LIN {X 0,Y 762.34,Z 876.166,A -85,B 0,C 180,E1 608.123,E2 608.123} C_VEL
LIN {X 0,Y 762.229,Z 909.531,A -85,B 0,C 180,E1 610.705,E2 610.705} C_VEL
LIN {X 0,Y 762.052,Z 938.578,A -85,B 0,C 180,E1 613.544,E2 613.544} C_VEL
LIN {X 0,Y 761.987,Z 962.68,A -85,B 0,C 180,E1 616.554,E2 616.554} C_VEL
LIN {X 0,Y 761.986,Z 981.631,A -85,B 0,C 180,E1 619.694,E2 619.694} C_VEL
LIN {X 0,Y 761.996,Z 994.243,A -85,B 0,C 180,E1 622.577,E2 622.577} C_VEL
LIN {X 0,Y 761.971,Z 1003.667,A -85,B 0,C 180,E1 626.012,E2 626.012} C_VEL
LIN {X 0,Y 762.065,Z 1007.172,A -85,B 0,C 180,E1 628.864,E2 628.864} C_VEL
LIN {X 0,Y 762.131,Z 1006.217,A -85,B 0,C 180,E1 632.282,E2 632.282} C_VEL
LIN {X 0,Y 762.103,Z 999.625,A -85,B 0,C 180,E1 635.708,E2 635.708} C_VEL
LIN {X 0,Y 762.107,Z 988.509,A -85,B 0,C 180,E1 638.867,E2 638.867} C_VEL
LIN {X 0,Y 762.098,Z 970.007,A -85,B 0,C 180,E1 642.344,E2 642.344} C_VEL
LIN {X 0,Y 762.102,Z 946.3,A -85,B 0,C 180,E1 645.573,E2 645.573} C_VEL
LIN {X 0,Y 762.212,Z 919.441,A -85,B 0,C 180,E1 648.399,E2 648.399} C_VEL
LIN {X 0,Y 762.327,Z 887.292,A -85,B 0,C 180,E1 651.08,E2 651.08} C_VEL
LIN {X 0,Y 762.452,Z 851.896,A -85,B 0,C 180,E1 653.423,E2 653.423} C_VEL
LIN {X 0,Y 762.604,Z 810.86,A -85,B 0,C 180,E1 655.528,E2 655.528} C_VEL
LIN {X 0,Y 762.736,Z 768.716,A -85,B 0,C 180,E1 657.14,E2 657.14} C_VEL
LIN {X 0,Y 762.819,Z 726.885,A -85,B 0,C 180,E1 658.273,E2 658.273} C_VEL
LIN {X 0,Y 762.768,Z 682.925,A -85,B 0,C 180,E1 659,E2 659} C_VEL
LIN {X 0,Y 761.872,Z 606.141,A -85,B 0,C 180,E1 659.857,E2 659.857} C_VEL
LIN {X 0,Y 761.765,Z 601.31,A -85,B 0,C 180,E1 659.987,E2 659.987} C_VEL
LIN {X 0,Y 761.618,Z 601.31,A -85,B 0,C 180,E1 663.856,E2 663.856} C_VEL
LIN {X 0,Y 761.749,Z 601.31,A -85,B 0,C 180,E1 668.074,E2 668.074} C_VEL
LIN {X 0,Y 761.892,Z 601.31,A -85,B 0,C 180,E1 672.633,E2 672.633} C_VEL
LIN {X 0,Y 761.767,Z 601.31,A -85,B 0,C 180,E1 675.889,E2 675.889} C_VEL
LIN {X 0,Y 761.89,Z 601.31,A -85,B 0,C 180,E1 680.865,E2 680.865} C_VEL
LIN {X 0,Y 761.687,Z 601.31,A -85,B 0,C 180,E1 686.158,E2 686.158} C_VEL
LIN {X 0,Y 761.768,Z 601.31,A -85,B 0,C 180,E1 690.186,E2 690.186} C_VEL
LIN {X 0,Y 761.993,Z 601.31,A -85,B 0,C 180,E1 694.062,E2 694.062} C_VEL
LIN {X 0,Y 762.103,Z 601.31,A -85,B 0,C 180,E1 697.809,E2 697.809} C_VEL
LIN {X 0,Y 761.881,Z 601.31,A -85,B 0,C 180,E1 702.681,E2 702.681} C_VEL
LIN {X 0,Y 761.587,Z 601.31,A -85,B 0,C 180,E1 707.36,E2 707.36} C_VEL
LIN {X 0,Y 761.764,Z 601.31,A -85,B 0,C 180,E1 710.844,E2 710.844} C_VEL
LIN {X 0,Y 761.847,Z 601.31,A -85,B 0,C 180,E1 714.293,E2 714.293} C_VEL
LIN {X 0,Y 761.764,Z 601.31,A -85,B 0,C 180,E1 718.859,E2 718.859} C_VEL
LIN {X 0,Y 761.801,Z 601.31,A -85,B 0,C 180,E1 722.278,E2 722.278} C_VEL
LIN {X 0,Y 761.796,Z 601.31,A -85,B 0,C 180,E1 725.985,E2 725.985} C_VEL
LIN {X 0,Y 761.725,Z 601.31,A -85,B 0,C 180,E1 730.309,E2 730.309} C_VEL
LIN {X 0,Y 761.689,Z 601.31,A -85,B 0,C 180,E1 733.806,E2 733.806} C_VEL
LIN {X 0,Y 761.794,Z 601.31,A -85,B 0,C 180,E1 737.353,E2 737.353} C_VEL
LIN {X 0,Y 761.769,Z 601.31,A -85,B 0,C 180,E1 740.973,E2 740.973} C_VEL
LIN {X 0,Y 761.784,Z 601.31,A -85,B 0,C 180,E1 744.682,E2 744.682} C_VEL
LIN {X 0,Y 761.75,Z 601.31,A -85,B 0,C 180,E1 748.924,E2 748.924} C_VEL
LIN {X 0,Y 761.669,Z 601.31,A -85,B 0,C 180,E1 753.325,E2 753.325} C_VEL
LIN {X 0,Y 761.815,Z 601.31,A -85,B 0,C 180,E1 758.055,E2 758.055} C_VEL
LIN {X 0,Y 761.92,Z 601.31,A -85,B 0,C 180,E1 762.62,E2 762.62} C_VEL
LIN {X 0,Y 761.8,Z 601.31,A -85,B 0,C 180,E1 765.877,E2 765.877} C_VEL
LIN {X 0,Y 761.888,Z 601.31,A -85,B 0,C 180,E1 770.843,E2 770.843} C_VEL
LIN {X 0,Y 761.695,Z 601.31,A -85,B 0,C 180,E1 776.148,E2 776.148} C_VEL
LIN {X 0,Y 761.797,Z 601.31,A -85,B 0,C 180,E1 780.178,E2 780.178} C_VEL
LIN {X 0,Y 762.041,Z 601.31,A -85,B 0,C 180,E1 784.056,E2 784.056} C_VEL
LIN {X 0,Y 762.028,Z 601.31,A -85,B 0,C 180,E1 787.26,E2 787.26} C_VEL
LIN {X 0,Y 762.54,Z 645.779,A -85,B 0,C 180,E1 788.084,E2 788.084} C_VEL
LIN {X 0,Y 762.458,Z 684.774,A -85,B 0,C 180,E1 789.266,E2 789.266} C_VEL
LIN {X 0,Y 762.403,Z 722.656,A -85,B 0,C 180,E1 790.929,E2 790.929} C_VEL
LIN {X 0,Y 762.261,Z 757.459,A -85,B 0,C 180,E1 793.022,E2 793.022} C_VEL
LIN {X 0,Y 762.167,Z 786.299,A -85,B 0,C 180,E1 795.314,E2 795.314} C_VEL
LIN {X 0,Y 762.071,Z 810.258,A -85,B 0,C 180,E1 797.801,E2 797.801} C_VEL
LIN {X 0,Y 762.047,Z 828.293,A -85,B 0,C 180,E1 800.267,E2 800.267} C_VEL
LIN {X 0,Y 761.991,Z 843.361,A -85,B 0,C 180,E1 803.145,E2 803.145} C_VEL
LIN {X 0,Y 762.028,Z 852.817,A -85,B 0,C 180,E1 806.006,E2 806.006} C_VEL
LIN {X 0,Y 761.987,Z 857.117,A -85,B 0,C 180,E1 808.857,E2 808.857} C_VEL
LIN {X 0,Y 762.036,Z 857.043,A -85,B 0,C 180,E1 811.136,E2 811.136} C_VEL
LIN {X 0,Y 762.053,Z 852.609,A -85,B 0,C 180,E1 813.987,E2 813.987} C_VEL
LIN {X 0,Y 762.068,Z 843.027,A -85,B 0,C 180,E1 816.848,E2 816.848} C_VEL
LIN {X 0,Y 762.117,Z 827.787,A -85,B 0,C 180,E1 819.726,E2 819.726} C_VEL
LIN {X 0,Y 762.16,Z 805.811,A -85,B 0,C 180,E1 822.629,E2 822.629} C_VEL
LIN {X 0,Y 762.201,Z 780.366,A -85,B 0,C 180,E1 825.121,E2 825.121} C_VEL
LIN {X 0,Y 762.306,Z 750.674,A -85,B 0,C 180,E1 827.343,E2 827.343} C_VEL
LIN {X 0,Y 762.389,Z 717.941,A -85,B 0,C 180,E1 829.215,E2 829.215} C_VEL
LIN {X 0,Y 762.466,Z 681.392,A -85,B 0,C 180,E1 830.765,E2 830.765} C_VEL
LIN {X 0,Y 762.551,Z 643.878,A -85,B 0,C 180,E1 831.87,E2 831.87} C_VEL
LIN {X 0,Y 761.833,Z 605.111,A -85,B 0,C 180,E1 832.585,E2 832.585} C_VEL
LIN {X 0,Y 761.612,Z 601.31,A -85,B 0,C 180,E1 832.669,E2 832.669} C_VEL
LIN {X 0,Y 761.644,Z 601.31,A -85,B 0,C 180,E1 837.226,E2 837.226} C_VEL
LIN {X 0,Y 761.976,Z 601.31,A -85,B 0,C 180,E1 842.469,E2 842.469} C_VEL
LIN {X 0,Y 761.746,Z 601.31,A -85,B 0,C 180,E1 848.066,E2 848.066} C_VEL
LIN {X 0,Y 761.932,Z 601.31,A -85,B 0,C 180,E1 852.641,E2 852.641} C_VEL
LIN {X 0,Y 761.805,Z 601.31,A -85,B 0,C 180,E1 855.896,E2 855.896} C_VEL
LIN {X 0,Y 761.868,Z 601.31,A -85,B 0,C 180,E1 860.857,E2 860.857} C_VEL
LIN {X 0,Y 761.724,Z 601.31,A -85,B 0,C 180,E1 866.163,E2 866.163} C_VEL
LIN {X 0,Y 761.776,Z 601.31,A -85,B 0,C 180,E1 870.19,E2 870.19} C_VEL
LIN {X 0,Y 762.023,Z 601.31,A -85,B 0,C 180,E1 874.066,E2 874.066} C_VEL
LIN {X 0,Y 762.052,Z 601.31,A -85,B 0,C 180,E1 877.81,E2 877.81} C_VEL
LIN {X 0,Y 761.635,Z 601.31,A -85,B 0,C 180,E1 883.09,E2 883.09} C_VEL
LIN {X 0,Y 761.273,Z 601.31,A -85,B 0,C 180,E1 883.156,E2 883.156} C_VEL
LIN {X 0,Y 762.323,Z 623.556,A -85,B 0,C 180,E1 883.403,E2 883.403} C_VEL
LIN {X 0,Y 762.406,Z 691.577,A -85,B 0,C 180,E1 884.146,E2 884.146} C_VEL
LIN {X 0,Y 762.394,Z 725.928,A -85,B 0,C 180,E1 884.995,E2 884.995} C_VEL
LIN {X 0,Y 762.322,Z 757.575,A -85,B 0,C 180,E1 886.262,E2 886.262} C_VEL
LIN {X 0,Y 762.237,Z 786.773,A -85,B 0,C 180,E1 887.957,E2 887.957} C_VEL
LIN {X 0,Y 762.177,Z 811.663,A -85,B 0,C 180,E1 889.986,E2 889.986} C_VEL
LIN {X 0,Y 762.127,Z 830.612,A -85,B 0,C 180,E1 892.147,E2 892.147} C_VEL
LIN {X 0,Y 762.134,Z 843.351,A -85,B 0,C 180,E1 894.211,E2 894.211} C_VEL
LIN {X 0,Y 758.218,Z 848.975,A -85,B 0,C 180,E1 895.428,E2 895.428} C_VEL
LIN {X 0,Y 754.212,Z 853.071,A -85,B 0,C 180,E1 896.691,E2 896.691} C_VEL
LIN {X 0,Y 754.206,Z 856.957,A -85,B 0,C 180,E1 898.851,E2 898.851} C_VEL
LIN {X 0,Y 754.232,Z 856.876,A -85,B 0,C 180,E1 901.152,E2 901.152} C_VEL
LIN {X 0,Y 754.27,Z 852.443,A -85,B 0,C 180,E1 903.456,E2 903.456} C_VEL
LIN {X 0,Y 754.27,Z 841.701,A -85,B 0,C 180,E1 906.072,E2 906.072} C_VEL
LIN {X 0,Y 754.302,Z 825.438,A -85,B 0,C 180,E1 908.519,E2 908.519} C_VEL
LIN {X 0,Y 754.383,Z 804.377,A -85,B 0,C 180,E1 910.706,E2 910.706} C_VEL
LIN {X 0,Y 754.485,Z 778.727,A -85,B 0,C 180,E1 912.614,E2 912.614} C_VEL
LIN {X 0,Y 754.602,Z 749.589,A -85,B 0,C 180,E1 914.164,E2 914.164} C_VEL
LIN {X 0,Y 754.72,Z 717.18,A -85,B 0,C 180,E1 915.339,E2 915.339} C_VEL
LIN {X 0,Y 754.8,Z 683.929,A -85,B 0,C 180,E1 916.051,E2 916.051} C_VEL
LIN {X 0,Y 754.166,Z 601.31,A -85,B 0,C 180,E1 916.936,E2 916.936} C_VEL
LIN {X 0,Y 753.78,Z 601.31,A -85,B 0,C 180,E1 921.209,E2 921.209} C_VEL
LIN {X 0,Y 753.771,Z 601.31,A -85,B 0,C 180,E1 925.241,E2 925.241} C_VEL
LIN {X 0,Y 753.87,Z 601.31,A -85,B 0,C 180,E1 928.836,E2 928.836} C_VEL
LIN {X 0,Y 753.932,Z 601.31,A -85,B 0,C 180,E1 932.857,E2 932.857} C_VEL
LIN {X 0,Y 754.133,Z 601.31,A -85,B 0,C 180,E1 937.06,E2 937.06} C_VEL
LIN {X 0,Y 753.998,Z 601.31,A -85,B 0,C 180,E1 943.089,E2 943.089} C_VEL
LIN {X 0,Y 753.625,Z 601.31,A -85,B 0,C 180,E1 946.88,E2 946.88} C_VEL
LIN {X 0,Y 753.748,Z 601.31,A -85,B 0,C 180,E1 951.614,E2 951.614} C_VEL
LIN {X 0,Y 753.721,Z 601.31,A -85,B 0,C 180,E1 955.748,E2 955.748} C_VEL
LIN {X 0,Y 753.863,Z 601.885,A -85,B 0,C 180,E1 959.747,E2 959.747} C_VEL
LIN {X 0,Y 755.848,Z 628.178,A -85,B 0,C 180,E1 960.118,E2 960.118} C_VEL
LIN {X 0,Y 755.868,Z 706.435,A -85,B 0,C 180,E1 961.047,E2 961.047} C_VEL
LIN {X 0,Y 755.568,Z 749.174,A -85,B 0,C 180,E1 961.985,E2 961.985} C_VEL
LIN {X 0,Y 755.392,Z 793.596,A -85,B 0,C 180,E1 963.474,E2 963.474} C_VEL
LIN {X 0,Y 755.115,Z 836.094,A -85,B 0,C 180,E1 965.447,E2 965.447} C_VEL
LIN {X 0,Y 754.819,Z 873.88,A -85,B 0,C 180,E1 967.738,E2 967.738} C_VEL
LIN {X 0,Y 754.581,Z 907.463,A -85,B 0,C 180,E1 970.322,E2 970.322} C_VEL
LIN {X 0,Y 754.32,Z 936,A -85,B 0,C 180,E1 973.081,E2 973.081} C_VEL
LIN {X 0,Y 754.175,Z 961.574,A -85,B 0,C 180,E1 976.246,E2 976.246} C_VEL
LIN {X 0,Y 754.119,Z 981.632,A -85,B 0,C 180,E1 979.585,E2 979.585} C_VEL
LIN {X 0,Y 754.142,Z 994.243,A -85,B 0,C 180,E1 982.499,E2 982.499} C_VEL
LIN {X 0,Y 754.09,Z 1003.668,A -85,B 0,C 180,E1 985.97,E2 985.97} C_VEL
LIN {X 0,Y 754.162,Z 1007.172,A -85,B 0,C 180,E1 988.852,E2 988.852} C_VEL
LIN {X 0,Y 754.224,Z 1006.217,A -85,B 0,C 180,E1 992.306,E2 992.306} C_VEL
LIN {X 0,Y 754.209,Z 999.625,A -85,B 0,C 180,E1 995.768,E2 995.768} C_VEL
LIN {X 0,Y 754.2,Z 988.508,A -85,B 0,C 180,E1 998.961,E2 998.961} C_VEL
LIN {X 0,Y 754.225,Z 970.008,A -85,B 0,C 180,E1 1002.475,E2 1002.475} C_VEL
LIN {X 0,Y 754.305,Z 947.009,A -85,B 0,C 180,E1 1005.651,E2 1005.651} C_VEL
LIN {X 0,Y 754.494,Z 919.44,A -85,B 0,C 180,E1 1008.594,E2 1008.594} C_VEL
LIN {X 0,Y 754.718,Z 887.799,A -85,B 0,C 180,E1 1011.265,E2 1011.265} C_VEL
LIN {X 0,Y 755.02,Z 851.9,A -85,B 0,C 180,E1 1013.667,E2 1013.667} C_VEL
LIN {X 0,Y 755.34,Z 809.958,A -85,B 0,C 180,E1 1015.834,E2 1015.834} C_VEL
LIN {X 0,Y 755.646,Z 767.167,A -85,B 0,C 180,E1 1017.468,E2 1017.468} C_VEL
LIN {X 0,Y 755.842,Z 726.268,A -85,B 0,C 180,E1 1018.57,E2 1018.57} C_VEL
LIN {X 0,Y 755.849,Z 682.925,A -85,B 0,C 180,E1 1019.291,E2 1019.291} C_VEL
LIN {X 0,Y 755.032,Z 606.95,A -85,B 0,C 180,E1 1020.146,E2 1020.146} C_VEL
LIN {X 0,Y 754.118,Z 601.31,A -85,B 0,C 180,E1 1020.252,E2 1020.252} C_VEL
LIN {X 0,Y 753.632,Z 601.31,A -85,B 0,C 180,E1 1024.496,E2 1024.496} C_VEL
LIN {X 0,Y 753.757,Z 601.31,A -85,B 0,C 180,E1 1028.387,E2 1028.387} C_VEL
LIN {X 0,Y 754.007,Z 601.31,A -85,B 0,C 180,E1 1033.672,E2 1033.672} C_VEL
LIN {X 0,Y 753.581,Z 601.31,A -85,B 0,C 180,E1 1038.44,E2 1038.44} C_VEL
LIN {X 0,Y 753.63,Z 601.31,A -85,B 0,C 180,E1 1042.911,E2 1042.911} C_VEL
LIN {X 0,Y 753.695,Z 601.31,A -85,B 0,C 180,E1 1047.609,E2 1047.609} C_VEL
LIN {X 0,Y 753.729,Z 601.31,A -85,B 0,C 180,E1 1052.199,E2 1052.199} C_VEL
LIN {X 0,Y 753.819,Z 601.31,A -85,B 0,C 180,E1 1056.3,E2 1056.3} C_VEL
LIN {X 0,Y 753.71,Z 601.31,A -85,B 0,C 180,E1 1060.019,E2 1060.019} C_VEL
LIN {X 0,Y 753.885,Z 601.31,A -85,B 0,C 180,E1 1063.659,E2 1063.659} C_VEL
LIN {X 0,Y 753.75,Z 601.31,A -85,B 0,C 180,E1 1068.404,E2 1068.404} C_VEL
LIN {X 0,Y 754.071,Z 601.31,A -85,B 0,C 180,E1 1073.075,E2 1073.075} C_VEL
LIN {X 0,Y 754.069,Z 601.31,A -85,B 0,C 180,E1 1077.696,E2 1077.696} C_VEL
LIN {X 0,Y 753.907,Z 601.31,A -85,B 0,C 180,E1 1082.302,E2 1082.302} C_VEL
LIN {X 0,Y 753.928,Z 601.31,A -85,B 0,C 180,E1 1085.765,E2 1085.765} C_VEL
LIN {X 0,Y 753.847,Z 601.31,A -85,B 0,C 180,E1 1089.957,E2 1089.957} C_VEL
LIN {X 0,Y 753.782,Z 601.31,A -85,B 0,C 180,E1 1093.954,E2 1093.954} C_VEL
LIN {X 0,Y 753.864,Z 601.31,A -85,B 0,C 180,E1 1097.542,E2 1097.542} C_VEL
LIN {X 0,Y 753.831,Z 601.31,A -85,B 0,C 180,E1 1101.205,E2 1101.205} C_VEL
LIN {X 0,Y 753.786,Z 601.31,A -85,B 0,C 180,E1 1105.229,E2 1105.229} C_VEL
LIN {X 0,Y 753.885,Z 601.31,A -85,B 0,C 180,E1 1108.832,E2 1108.832} C_VEL
LIN {X 0,Y 753.931,Z 601.31,A -85,B 0,C 180,E1 1112.853,E2 1112.853} C_VEL
LIN {X 0,Y 754.136,Z 601.31,A -85,B 0,C 180,E1 1117.057,E2 1117.057} C_VEL
LIN {X 0,Y 753.978,Z 601.31,A -85,B 0,C 180,E1 1123.086,E2 1123.086} C_VEL
LIN {X 0,Y 753.619,Z 601.31,A -85,B 0,C 180,E1 1126.871,E2 1126.871} C_VEL
LIN {X 0,Y 753.752,Z 601.31,A -85,B 0,C 180,E1 1131.609,E2 1131.609} C_VEL
LIN {X 0,Y 753.757,Z 601.31,A -85,B 0,C 180,E1 1135.743,E2 1135.743} C_VEL
LIN {X 0,Y 753.894,Z 601.31,A -85,B 0,C 180,E1 1139.834,E2 1139.834} C_VEL
LIN {X 0,Y 753.94,Z 601.31,A -85,B 0,C 180,E1 1145.033,E2 1145.033} C_VEL
LIN {X 0,Y 754.109,Z 601.31,A -85,B 0,C 180,E1 1147.024,E2 1147.024} C_VEL
LIN {X 0,Y 755.192,Z 640.857,A -85,B 0,C 180,E1 1147.743,E2 1147.743} C_VEL
LIN {X 0,Y 754.968,Z 679.523,A -85,B 0,C 180,E1 1148.86,E2 1148.86} C_VEL
LIN {X 0,Y 754.83,Z 715.918,A -85,B 0,C 180,E1 1150.393,E2 1150.393} C_VEL
LIN {X 0,Y 754.617,Z 750.094,A -85,B 0,C 180,E1 1152.346,E2 1152.346} C_VEL
LIN {X 0,Y 754.464,Z 780.517,A -85,B 0,C 180,E1 1154.642,E2 1154.642} C_VEL
LIN {X 0,Y 754.323,Z 806.573,A -85,B 0,C 180,E1 1157.232,E2 1157.232} C_VEL
LIN {X 0,Y 754.194,Z 827.885,A -85,B 0,C 180,E1 1160.096,E2 1160.096} C_VEL
LIN {X 0,Y 754.105,Z 843.357,A -85,B 0,C 180,E1 1163.073,E2 1163.073} C_VEL
LIN {X 0,Y 754.138,Z 852.811,A -85,B 0,C 180,E1 1165.964,E2 1165.964} C_VEL
LIN {X 0,Y 754.088,Z 857.117,A -85,B 0,C 180,E1 1168.845,E2 1168.845} C_VEL
LIN {X 0,Y 754.135,Z 857.044,A -85,B 0,C 180,E1 1171.148,E2 1171.148} C_VEL
LIN {X 0,Y 754.165,Z 852.612,A -85,B 0,C 180,E1 1174.029,E2 1174.029} C_VEL
LIN {X 0,Y 754.174,Z 843.026,A -85,B 0,C 180,E1 1176.92,E2 1176.92} C_VEL
LIN {X 0,Y 754.26,Z 826.849,A -85,B 0,C 180,E1 1179.976,E2 1179.976} C_VEL
LIN {X 0,Y 754.353,Z 805.82,A -85,B 0,C 180,E1 1182.761,E2 1182.761} C_VEL
LIN {X 0,Y 754.477,Z 779.502,A -85,B 0,C 180,E1 1185.354,E2 1185.354} C_VEL
LIN {X 0,Y 754.675,Z 749.623,A -85,B 0,C 180,E1 1187.594,E2 1187.594} C_VEL
LIN {X 0,Y 754.821,Z 716.321,A -85,B 0,C 180,E1 1189.497,E2 1189.497} C_VEL
LIN {X 0,Y 755.016,Z 679.284,A -85,B 0,C 180,E1 1191.057,E2 1191.057} C_VEL
LIN {X 0,Y 755.2,Z 640.623,A -85,B 0,C 180,E1 1192.172,E2 1192.172} C_VEL
LIN {X 0,Y 754.253,Z 603.48,A -85,B 0,C 180,E1 1192.845,E2 1192.845} C_VEL
LIN {X 0,Y 754.25,Z 601.31,A -85,B 0,C 180,E1 1192.903,E2 1192.903} C_VEL
LIN {X 0,Y 753.868,Z 601.31,A -85,B 0,C 180,E1 1198.837,E2 1198.837} C_VEL
LIN {X 0,Y 753.95,Z 601.31,A -85,B 0,C 180,E1 1202.858,E2 1202.858} C_VEL
LIN {X 0,Y 754.077,Z 601.31,A -85,B 0,C 180,E1 1207.067,E2 1207.067} C_VEL
LIN {X 0,Y 753.989,Z 601.31,A -85,B 0,C 180,E1 1213.094,E2 1213.094} C_VEL
LIN {X 0,Y 753.624,Z 601.31,A -85,B 0,C 180,E1 1216.889,E2 1216.889} C_VEL
LIN {X 0,Y 753.735,Z 601.31,A -85,B 0,C 180,E1 1221.623,E2 1221.623} C_VEL
LIN {X 0,Y 753.782,Z 601.31,A -85,B 0,C 180,E1 1225.758,E2 1225.758} C_VEL
LIN {X 0,Y 753.875,Z 601.31,A -85,B 0,C 180,E1 1229.845,E2 1229.845} C_VEL
LIN {X 0,Y 753.931,Z 601.31,A -85,B 0,C 180,E1 1234.733,E2 1234.733} C_VEL
LIN {X 0,Y 753.75,Z 601.31,A -85,B 0,C 180,E1 1238.793,E2 1238.793} C_VEL
LIN {X 0,Y 753.745,Z 601.31,A -85,B 0,C 180,E1 1242.982,E2 1242.982} C_VEL
LIN {X 0,Y 754.764,Z 636.829,A -85,B 0,C 180,E1 1243.362,E2 1243.362} C_VEL
LIN {X 0,Y 754.82,Z 691.297,A -85,B 0,C 180,E1 1243.978,E2 1243.978} C_VEL
LIN {X 0,Y 754.731,Z 725.142,A -85,B 0,C 180,E1 1244.815,E2 1244.815} C_VEL
LIN {X 0,Y 754.602,Z 756.393,A -85,B 0,C 180,E1 1246.062,E2 1246.062} C_VEL
LIN {X 0,Y 754.477,Z 784.673,A -85,B 0,C 180,E1 1247.684,E2 1247.684} C_VEL
LIN {X 0,Y 754.34,Z 809.763,A -85,B 0,C 180,E1 1249.694,E2 1249.694} C_VEL
LIN {X 0,Y 754.252,Z 829.664,A -85,B 0,C 180,E1 1251.939,E2 1251.939} C_VEL
LIN {X 0,Y 754.257,Z 843.806,A -85,B 0,C 180,E1 1254.238,E2 1254.238} C_VEL
LIN {X 0,Y 754.212,Z 853.071,A -85,B 0,C 180,E1 1256.691,E2 1256.691} C_VEL
LIN {X 0,Y 750.206,Z 855.873,A -85,B 0,C 180,E1 1257.968,E2 1257.968} C_VEL
LIN {X 0,Y 746.264,Z 857.157,A -85,B 0,C 180,E1 1259.272,E2 1259.272} C_VEL
LIN {X 0,Y 746.329,Z 856.877,A -85,B 0,C 180,E1 1261.165,E2 1261.165} C_VEL
LIN {X 0,Y 746.368,Z 852.443,A -85,B 0,C 180,E1 1263.492,E2 1263.492} C_VEL
LIN {X 0,Y 746.4,Z 841.954,A -85,B 0,C 180,E1 1266.089,E2 1266.089} C_VEL
LIN {X 0,Y 746.455,Z 825.442,A -85,B 0,C 180,E1 1268.609,E2 1268.609} C_VEL
LIN {X 0,Y 746.555,Z 804.383,A -85,B 0,C 180,E1 1270.82,E2 1270.82} C_VEL
LIN {X 0,Y 746.756,Z 778.737,A -85,B 0,C 180,E1 1272.746,E2 1272.746} C_VEL
LIN {X 0,Y 746.896,Z 749.605,A -85,B 0,C 180,E1 1274.313,E2 1274.313} C_VEL
LIN {X 0,Y 747.098,Z 717.199,A -85,B 0,C 180,E1 1275.499,E2 1275.499} C_VEL
LIN {X 0,Y 747.235,Z 682.659,A -85,B 0,C 180,E1 1276.238,E2 1276.238} C_VEL
LIN {X 0,Y 746.309,Z 602.53,A -85,B 0,C 180,E1 1277.08,E2 1277.08} C_VEL
LIN {X 0,Y 746.228,Z 601.31,A -85,B 0,C 180,E1 1277.159,E2 1277.159} C_VEL
LIN {X 0,Y 745.865,Z 601.31,A -85,B 0,C 180,E1 1281.445,E2 1281.445} C_VEL
LIN {X 0,Y 745.893,Z 601.31,A -85,B 0,C 180,E1 1285.247,E2 1285.247} C_VEL
LIN {X 0,Y 745.916,Z 601.31,A -85,B 0,C 180,E1 1289.173,E2 1289.173} C_VEL
LIN {X 0,Y 745.85,Z 601.31,A -85,B 0,C 180,E1 1293.606,E2 1293.606} C_VEL
LIN {X 0,Y 746.058,Z 601.31,A -85,B 0,C 180,E1 1297.626,E2 1297.626} C_VEL
LIN {X 0,Y 746.135,Z 601.31,A -85,B 0,C 180,E1 1303.656,E2 1303.656} C_VEL
LIN {X 0,Y 745.689,Z 601.31,A -85,B 0,C 180,E1 1308.737,E2 1308.737} C_VEL
LIN {X 0,Y 745.709,Z 601.31,A -85,B 0,C 180,E1 1312.446,E2 1312.446} C_VEL
LIN {X 0,Y 745.663,Z 601.31,A -85,B 0,C 180,E1 1316.73,E2 1316.73} C_VEL
LIN {X 0,Y 746.053,Z 601.31,A -85,B 0,C 180,E1 1319.375,E2 1319.375} C_VEL
LIN {X 0,Y 748.965,Z 625.546,A -85,B 0,C 180,E1 1319.786,E2 1319.786} C_VEL
LIN {X 0,Y 748.943,Z 707.238,A -85,B 0,C 180,E1 1320.767,E2 1320.767} C_VEL
LIN {X 0,Y 748.513,Z 750.506,A -85,B 0,C 180,E1 1321.737,E2 1321.737} C_VEL
LIN {X 0,Y 748.177,Z 794.938,A -85,B 0,C 180,E1 1323.253,E2 1323.253} C_VEL
LIN {X 0,Y 747.729,Z 838.22,A -85,B 0,C 180,E1 1325.3,E2 1325.3} C_VEL
LIN {X 0,Y 747.242,Z 878.449,A -85,B 0,C 180,E1 1327.814,E2 1327.814} C_VEL
LIN {X 0,Y 746.838,Z 914.108,A -85,B 0,C 180,E1 1330.699,E2 1330.699} C_VEL
LIN {X 0,Y 746.499,Z 943.919,A -85,B 0,C 180,E1 1333.797,E2 1333.797} C_VEL
LIN {X 0,Y 746.258,Z 967.593,A -85,B 0,C 180,E1 1337.01,E2 1337.01} C_VEL
LIN {X 0,Y 746.242,Z 983.572,A -85,B 0,C 180,E1 1339.86,E2 1339.86} C_VEL
LIN {X 0,Y 746.172,Z 996.17,A -85,B 0,C 180,E1 1343.005,E2 1343.005} C_VEL
LIN {X 0,Y 746.214,Z 1003.668,A -85,B 0,C 180,E1 1345.928,E2 1345.928} C_VEL
LIN {X 0,Y 746.26,Z 1007.172,A -85,B 0,C 180,E1 1348.84,E2 1348.84} C_VEL
LIN {X 0,Y 746.317,Z 1006.217,A -85,B 0,C 180,E1 1352.33,E2 1352.33} C_VEL
LIN {X 0,Y 746.284,Z 999.397,A -85,B 0,C 180,E1 1355.915,E2 1355.915} C_VEL
LIN {X 0,Y 746.254,Z 987.165,A -85,B 0,C 180,E1 1359.351,E2 1359.351} C_VEL
LIN {X 0,Y 746.349,Z 970.009,A -85,B 0,C 180,E1 1362.609,E2 1362.609} C_VEL
LIN {X 0,Y 746.476,Z 946.303,A -85,B 0,C 180,E1 1365.907,E2 1365.907} C_VEL
LIN {X 0,Y 746.766,Z 919.441,A -85,B 0,C 180,E1 1368.794,E2 1368.794} C_VEL
LIN {X 0,Y 747.144,Z 887.8,A -85,B 0,C 180,E1 1371.491,E2 1371.491} C_VEL
LIN {X 0,Y 747.614,Z 850.385,A -85,B 0,C 180,E1 1374.004,E2 1374.004} C_VEL
LIN {X 0,Y 748.081,Z 809.815,A -85,B 0,C 180,E1 1376.11,E2 1376.11} C_VEL
LIN {X 0,Y 748.539,Z 767.171,A -85,B 0,C 180,E1 1377.751,E2 1377.751} C_VEL
LIN {X 0,Y 748.866,Z 727.001,A -85,B 0,C 180,E1 1378.846,E2 1378.846} C_VEL
LIN {X 0,Y 748.972,Z 682.697,A -85,B 0,C 180,E1 1379.589,E2 1379.589} C_VEL
LIN {X 0,Y 748.199,Z 607.511,A -85,B 0,C 180,E1 1380.445,E2 1380.445} C_VEL
LIN {X 0,Y 746.174,Z 601.31,A -85,B 0,C 180,E1 1380.634,E2 1380.634} C_VEL
LIN {X 0,Y 745.874,Z 601.31,A -85,B 0,C 180,E1 1386.099,E2 1386.099} C_VEL
LIN {X 0,Y 745.816,Z 601.31,A -85,B 0,C 180,E1 1391.274,E2 1391.274} C_VEL
LIN {X 0,Y 746.03,Z 601.31,A -85,B 0,C 180,E1 1395.309,E2 1395.309} C_VEL
LIN {X 0,Y 745.867,Z 601.31,A -85,B 0,C 180,E1 1400.976,E2 1400.976} C_VEL
LIN {X 0,Y 745.786,Z 601.31,A -85,B 0,C 180,E1 1406.413,E2 1406.413} C_VEL
LIN {X 0,Y 745.814,Z 601.31,A -85,B 0,C 180,E1 1410.885,E2 1410.885} C_VEL
LIN {X 0,Y 746.009,Z 601.31,A -85,B 0,C 180,E1 1414.757,E2 1414.757} C_VEL
LIN {X 0,Y 745.903,Z 601.31,A -85,B 0,C 180,E1 1419.145,E2 1419.145} C_VEL
LIN {X 0,Y 745.978,Z 601.31,A -85,B 0,C 180,E1 1423.481,E2 1423.481} C_VEL
LIN {X 0,Y 745.83,Z 601.31,A -85,B 0,C 180,E1 1428.279,E2 1428.279} C_VEL
LIN {X 0,Y 746.16,Z 601.31,A -85,B 0,C 180,E1 1433.002,E2 1433.002} C_VEL
LIN {X 0,Y 746.166,Z 601.31,A -85,B 0,C 180,E1 1437.671,E2 1437.671} C_VEL
LIN {X 0,Y 746.005,Z 601.31,A -85,B 0,C 180,E1 1442.326,E2 1442.326} C_VEL
LIN {X 0,Y 746.017,Z 601.31,A -85,B 0,C 180,E1 1445.826,E2 1445.826} C_VEL
LIN {X 0,Y 745.924,Z 601.31,A -85,B 0,C 180,E1 1450.53,E2 1450.53} C_VEL
LIN {X 0,Y 746.045,Z 601.31,A -85,B 0,C 180,E1 1455.304,E2 1455.304} C_VEL
LIN {X 0,Y 745.98,Z 601.31,A -85,B 0,C 180,E1 1460.87,E2 1460.87} C_VEL
LIN {X 0,Y 745.908,Z 601.31,A -85,B 0,C 180,E1 1465.244,E2 1465.244} C_VEL
LIN {X 0,Y 745.92,Z 601.31,A -85,B 0,C 180,E1 1469.169,E2 1469.169} C_VEL
LIN {X 0,Y 745.842,Z 601.31,A -85,B 0,C 180,E1 1473.593,E2 1473.593} C_VEL
LIN {X 0,Y 746.05,Z 601.31,A -85,B 0,C 180,E1 1477.615,E2 1477.615} C_VEL
LIN {X 0,Y 746.106,Z 601.31,A -85,B 0,C 180,E1 1483.654,E2 1483.654} C_VEL
LIN {X 0,Y 745.718,Z 601.31,A -85,B 0,C 180,E1 1488.73,E2 1488.73} C_VEL
LIN {X 0,Y 745.73,Z 601.31,A -85,B 0,C 180,E1 1492.439,E2 1492.439} C_VEL
LIN {X 0,Y 745.76,Z 601.31,A -85,B 0,C 180,E1 1496.727,E2 1496.727} C_VEL
LIN {X 0,Y 745.824,Z 601.31,A -85,B 0,C 180,E1 1500.852,E2 1500.852} C_VEL
LIN {X 0,Y 746.109,Z 601.31,A -85,B 0,C 180,E1 1504.753,E2 1504.753} C_VEL
LIN {X 0,Y 746.156,Z 601.31,A -85,B 0,C 180,E1 1506.761,E2 1506.761} C_VEL
LIN {X 0,Y 747.817,Z 613.994,A -85,B 0,C 180,E1 1506.997,E2 1506.997} C_VEL
LIN {X 0,Y 747.823,Z 653.303,A -85,B 0,C 180,E1 1507.826,E2 1507.826} C_VEL
LIN {X 0,Y 747.52,Z 692.203,A -85,B 0,C 180,E1 1509.124,E2 1509.124} C_VEL
LIN {X 0,Y 747.171,Z 727.649,A -85,B 0,C 180,E1 1510.799,E2 1510.799} C_VEL
LIN {X 0,Y 746.852,Z 759.517,A -85,B 0,C 180,E1 1512.811,E2 1512.811} C_VEL
LIN {X 0,Y 746.6,Z 787.893,A -85,B 0,C 180,E1 1515.151,E2 1515.151} C_VEL
LIN {X 0,Y 746.414,Z 811.47,A -85,B 0,C 180,E1 1517.69,E2 1517.69} C_VEL
LIN {X 0,Y 746.271,Z 830.554,A -85,B 0,C 180,E1 1520.441,E2 1520.441} C_VEL
LIN {X 0,Y 746.2,Z 844.614,A -85,B 0,C 180,E1 1523.321,E2 1523.321} C_VEL
LIN {X 0,Y 746.257,Z 852.804,A -85,B 0,C 180,E1 1525.922,E2 1525.922} C_VEL
LIN {X 0,Y 746.189,Z 857.115,A -85,B 0,C 180,E1 1528.833,E2 1528.833} C_VEL
LIN {X 0,Y 746.235,Z 857.044,A -85,B 0,C 180,E1 1531.16,E2 1531.16} C_VEL
LIN {X 0,Y 746.286,Z 852.609,A -85,B 0,C 180,E1 1534.072,E2 1534.072} C_VEL
LIN {X 0,Y 746.3,Z 843.025,A -85,B 0,C 180,E1 1536.994,E2 1536.994} C_VEL
LIN {X 0,Y 746.406,Z 827.45,A -85,B 0,C 180,E1 1539.99,E2 1539.99} C_VEL
LIN {X 0,Y 746.533,Z 805.829,A -85,B 0,C 180,E1 1542.897,E2 1542.897} C_VEL
LIN {X 0,Y 746.715,Z 780.157,A -85,B 0,C 180,E1 1545.462,E2 1545.462} C_VEL
LIN {X 0,Y 746.973,Z 749.545,A -85,B 0,C 180,E1 1547.787,E2 1547.787} C_VEL
LIN {X 0,Y 747.27,Z 715.614,A -85,B 0,C 180,E1 1549.739,E2 1549.739} C_VEL
LIN {X 0,Y 747.581,Z 678.342,A -85,B 0,C 180,E1 1551.313,E2 1551.313} C_VEL
LIN {X 0,Y 747.87,Z 638.311,A -85,B 0,C 180,E1 1552.456,E2 1552.456} C_VEL
LIN {X 0,Y 747.007,Z 604.745,A -85,B 0,C 180,E1 1553.064,E2 1553.064} C_VEL
LIN {X 0,Y 746.302,Z 601.31,A -85,B 0,C 180,E1 1553.143,E2 1553.143} C_VEL
LIN {X 0,Y 745.901,Z 601.31,A -85,B 0,C 180,E1 1559.175,E2 1559.175} C_VEL
LIN {X 0,Y 745.868,Z 601.31,A -85,B 0,C 180,E1 1563.623,E2 1563.623} C_VEL
LIN {X 0,Y 745.985,Z 601.31,A -85,B 0,C 180,E1 1567.632,E2 1567.632} C_VEL
LIN {X 0,Y 746.116,Z 601.31,A -85,B 0,C 180,E1 1573.663,E2 1573.663} C_VEL
LIN {X 0,Y 745.744,Z 601.31,A -85,B 0,C 180,E1 1578.739,E2 1578.739} C_VEL
LIN {X 0,Y 745.718,Z 601.31,A -85,B 0,C 180,E1 1582.453,E2 1582.453} C_VEL
LIN {X 0,Y 745.773,Z 601.31,A -85,B 0,C 180,E1 1586.741,E2 1586.741} C_VEL
LIN {X 0,Y 745.812,Z 601.31,A -85,B 0,C 180,E1 1590.873,E2 1590.873} C_VEL
LIN {X 0,Y 746.04,Z 601.31,A -85,B 0,C 180,E1 1594.761,E2 1594.761} C_VEL
LIN {X 0,Y 745.757,Z 601.31,A -85,B 0,C 180,E1 1599.157,E2 1599.157} C_VEL
LIN {X 0,Y 746.186,Z 601.31,A -85,B 0,C 180,E1 1602.808,E2 1602.808} C_VEL
LIN {X 0,Y 747.185,Z 642.529,A -85,B 0,C 180,E1 1603.245,E2 1603.245} C_VEL
LIN {X 0,Y 747.207,Z 692.83,A -85,B 0,C 180,E1 1603.84,E2 1603.84} C_VEL
LIN {X 0,Y 747.071,Z 727.048,A -85,B 0,C 180,E1 1604.717,E2 1604.717} C_VEL
LIN {X 0,Y 746.867,Z 759.466,A -85,B 0,C 180,E1 1606.066,E2 1606.066} C_VEL
LIN {X 0,Y 746.669,Z 787.808,A -85,B 0,C 180,E1 1607.776,E2 1607.776} C_VEL
LIN {X 0,Y 746.498,Z 812.181,A -85,B 0,C 180,E1 1609.826,E2 1609.826} C_VEL
LIN {X 0,Y 746.419,Z 831.672,A -85,B 0,C 180,E1 1612.128,E2 1612.128} C_VEL
LIN {X 0,Y 746.359,Z 845.142,A -85,B 0,C 180,E1 1614.469,E2 1614.469} C_VEL
LIN {X 0,Y 746.27,Z 854.208,A -85,B 0,C 180,E1 1617.093,E2 1617.093} C_VEL
LIN {X 0,Y 746.264,Z 857.157,A -85,B 0,C 180,E1 1619.272,E2 1619.272} C_VEL
LIN {X 0,Y 743.738,Z 857.47,A -85,B 0,C 180,E1 1620.26,E2 1620.26} C_VEL
LIN {X 0,Y 738.392,Z 856.099,A -85,B 0,C 180,E1 1621.817,E2 1621.817} C_VEL
LIN {X 0,Y 738.369,Z 855.852,A -85,B 0,C 180,E1 1621.902,E2 1621.902} C_VEL
LIN {X 0,Y 738.465,Z 849.612,A -85,B 0,C 180,E1 1624.413,E2 1624.413} C_VEL
LIN {X 0,Y 738.517,Z 838.56,A -85,B 0,C 180,E1 1626.775,E2 1626.775} C_VEL
LIN {X 0,Y 738.606,Z 821.824,A -85,B 0,C 180,E1 1629.148,E2 1629.148} C_VEL
LIN {X 0,Y 738.783,Z 799.172,A -85,B 0,C 180,E1 1631.384,E2 1631.384} C_VEL
LIN {X 0,Y 739.04,Z 772.468,A -85,B 0,C 180,E1 1633.272,E2 1633.272} C_VEL
LIN {X 0,Y 739.29,Z 742.686,A -85,B 0,C 180,E1 1634.767,E2 1634.767} C_VEL
LIN {X 0,Y 739.548,Z 710.535,A -85,B 0,C 180,E1 1635.844,E2 1635.844} C_VEL
LIN {X 0,Y 739.649,Z 677.847,A -85,B 0,C 180,E1 1636.477,E2 1636.477} C_VEL
LIN {X 0,Y 738.772,Z 603.946,A -85,B 0,C 180,E1 1637.246,E2 1637.246} C_VEL
LIN {X 0,Y 738.295,Z 601.31,A -85,B 0,C 180,E1 1637.297,E2 1637.297} C_VEL
LIN {X 0,Y 737.95,Z 601.31,A -85,B 0,C 180,E1 1642.495,E2 1642.495} C_VEL
LIN {X 0,Y 737.96,Z 601.31,A -85,B 0,C 180,E1 1646.849,E2 1646.849} C_VEL
LIN {X 0,Y 738.036,Z 601.31,A -85,B 0,C 180,E1 1652.256,E2 1652.256} C_VEL
LIN {X 0,Y 738.041,Z 601.31,A -85,B 0,C 180,E1 1658.01,E2 1658.01} C_VEL
LIN {X 0,Y 738.121,Z 601.31,A -85,B 0,C 180,E1 1662.633,E2 1662.633} C_VEL
LIN {X 0,Y 737.776,Z 601.31,A -85,B 0,C 180,E1 1667.337,E2 1667.337} C_VEL
LIN {X 0,Y 737.824,Z 601.31,A -85,B 0,C 180,E1 1671.973,E2 1671.973} C_VEL
LIN {X 0,Y 737.809,Z 601.31,A -85,B 0,C 180,E1 1676.329,E2 1676.329} C_VEL
LIN {X 0,Y 738.057,Z 601.31,A -85,B 0,C 180,E1 1679.009,E2 1679.009} C_VEL
LIN {X 0,Y 741.163,Z 613.763,A -85,B 0,C 180,E1 1679.304,E2 1679.304} C_VEL
LIN {X 0,Y 742.176,Z 640.354,A -85,B 0,C 180,E1 1679.643,E2 1679.643} C_VEL
LIN {X 0,Y 741.973,Z 709.467,A -85,B 0,C 180,E1 1680.504,E2 1680.504} C_VEL
LIN {X 0,Y 741.454,Z 752.302,A -85,B 0,C 180,E1 1681.497,E2 1681.497} C_VEL
LIN {X 0,Y 740.975,Z 796.079,A -85,B 0,C 180,E1 1683.021,E2 1683.021} C_VEL
LIN {X 0,Y 740.352,Z 839.188,A -85,B 0,C 180,E1 1685.092,E2 1685.092} C_VEL
LIN {X 0,Y 739.723,Z 878.834,A -85,B 0,C 180,E1 1687.605,E2 1687.605} C_VEL
LIN {X 0,Y 739.166,Z 912.927,A -85,B 0,C 180,E1 1690.38,E2 1690.38} C_VEL
LIN {X 0,Y 738.71,Z 942.598,A -85,B 0,C 180,E1 1693.469,E2 1693.469} C_VEL
LIN {X 0,Y 738.435,Z 966.201,A -85,B 0,C 180,E1 1696.657,E2 1696.657} C_VEL
LIN {X 0,Y 738.361,Z 983.539,A -85,B 0,C 180,E1 1699.743,E2 1699.743} C_VEL
LIN {X 0,Y 738.283,Z 996.17,A -85,B 0,C 180,E1 1702.93,E2 1702.93} C_VEL
LIN {X 0,Y 738.316,Z 1003.668,A -85,B 0,C 180,E1 1705.884,E2 1705.884} C_VEL
LIN {X 0,Y 738.358,Z 1007.171,A -85,B 0,C 180,E1 1708.827,E2 1708.827} C_VEL
LIN {X 0,Y 738.427,Z 1006.218,A -85,B 0,C 180,E1 1712.355,E2 1712.355} C_VEL
LIN {X 0,Y 738.413,Z 999.626,A -85,B 0,C 180,E1 1715.892,E2 1715.892} C_VEL
LIN {X 0,Y 738.402,Z 988.507,A -85,B 0,C 180,E1 1719.154,E2 1719.154} C_VEL
LIN {X 0,Y 738.481,Z 970.01,A -85,B 0,C 180,E1 1722.746,E2 1722.746} C_VEL
LIN {X 0,Y 738.687,Z 946.305,A -85,B 0,C 180,E1 1726.079,E2 1726.079} C_VEL
LIN {X 0,Y 739.036,Z 919.442,A -85,B 0,C 180,E1 1728.998,E2 1728.998} C_VEL
LIN {X 0,Y 739.562,Z 887.842,A -85,B 0,C 180,E1 1731.72,E2 1731.72} C_VEL
LIN {X 0,Y 740.197,Z 850.389,A -85,B 0,C 180,E1 1734.26,E2 1734.26} C_VEL
LIN {X 0,Y 740.85,Z 809.342,A -85,B 0,C 180,E1 1736.406,E2 1736.406} C_VEL
LIN {X 0,Y 741.446,Z 767.174,A -85,B 0,C 180,E1 1738.039,E2 1738.039} C_VEL
LIN {X 0,Y 741.922,Z 726.074,A -85,B 0,C 180,E1 1739.162,E2 1739.162} C_VEL
LIN {X 0,Y 742.106,Z 682.502,A -85,B 0,C 180,E1 1739.893,E2 1739.893} C_VEL
LIN {X 0,Y 741.379,Z 609.729,A -85,B 0,C 180,E1 1740.73,E2 1740.73} C_VEL
LIN {X 0,Y 738.258,Z 601.31,A -85,B 0,C 180,E1 1740.998,E2 1740.998} C_VEL
LIN {X 0,Y 737.998,Z 601.31,A -85,B 0,C 180,E1 1746.815,E2 1746.815} C_VEL
LIN {X 0,Y 738.102,Z 601.31,A -85,B 0,C 180,E1 1752.648,E2 1752.648} C_VEL
LIN {X 0,Y 737.772,Z 601.31,A -85,B 0,C 180,E1 1757.342,E2 1757.342} C_VEL
LIN {X 0,Y 737.858,Z 601.31,A -85,B 0,C 180,E1 1761.979,E2 1761.979} C_VEL
LIN {X 0,Y 737.883,Z 601.31,A -85,B 0,C 180,E1 1766.335,E2 1766.335} C_VEL
LIN {X 0,Y 737.91,Z 601.31,A -85,B 0,C 180,E1 1770.48,E2 1770.48} C_VEL
LIN {X 0,Y 738.124,Z 601.31,A -85,B 0,C 180,E1 1774.592,E2 1774.592} C_VEL
LIN {X 0,Y 738.108,Z 601.31,A -85,B 0,C 180,E1 1778.318,E2 1778.318} C_VEL
LIN {X 0,Y 738.097,Z 601.31,A -85,B 0,C 180,E1 1783.3,E2 1783.3} C_VEL
LIN {X 0,Y 737.929,Z 601.31,A -85,B 0,C 180,E1 1788.152,E2 1788.152} C_VEL
LIN {X 0,Y 738.233,Z 601.31,A -85,B 0,C 180,E1 1792.926,E2 1792.926} C_VEL
LIN {X 0,Y 738.265,Z 601.31,A -85,B 0,C 180,E1 1797.646,E2 1797.646} C_VEL
LIN {X 0,Y 738.114,Z 601.31,A -85,B 0,C 180,E1 1802.351,E2 1802.351} C_VEL
LIN {X 0,Y 738.107,Z 601.31,A -85,B 0,C 180,E1 1805.889,E2 1805.889} C_VEL
LIN {X 0,Y 738.05,Z 601.31,A -85,B 0,C 180,E1 1810.644,E2 1810.644} C_VEL
LIN {X 0,Y 738.144,Z 601.31,A -85,B 0,C 180,E1 1815.472,E2 1815.472} C_VEL
LIN {X 0,Y 738.145,Z 601.31,A -85,B 0,C 180,E1 1820.418,E2 1820.418} C_VEL
LIN {X 0,Y 737.964,Z 601.31,A -85,B 0,C 180,E1 1825.535,E2 1825.535} C_VEL
LIN {X 0,Y 737.903,Z 601.31,A -85,B 0,C 180,E1 1830.404,E2 1830.404} C_VEL
LIN {X 0,Y 737.881,Z 601.31,A -85,B 0,C 180,E1 1835.087,E2 1835.087} C_VEL
LIN {X 0,Y 737.828,Z 601.31,A -85,B 0,C 180,E1 1839.528,E2 1839.528} C_VEL
LIN {X 0,Y 738.183,Z 601.31,A -85,B 0,C 180,E1 1844.244,E2 1844.244} C_VEL
LIN {X 0,Y 738.025,Z 601.31,A -85,B 0,C 180,E1 1850.468,E2 1850.468} C_VEL
LIN {X 0,Y 737.955,Z 601.31,A -85,B 0,C 180,E1 1855.195,E2 1855.195} C_VEL
LIN {X 0,Y 737.931,Z 601.31,A -85,B 0,C 180,E1 1860.472,E2 1860.472} C_VEL
LIN {X 0,Y 738.195,Z 601.31,A -85,B 0,C 180,E1 1864.544,E2 1864.544} C_VEL
LIN {X 0,Y 738.239,Z 601.31,A -85,B 0,C 180,E1 1866.51,E2 1866.51} C_VEL
LIN {X 0,Y 740.509,Z 611.719,A -85,B 0,C 180,E1 1866.721,E2 1866.721} C_VEL
LIN {X 0,Y 740.449,Z 653.277,A -85,B 0,C 180,E1 1867.593,E2 1867.593} C_VEL
LIN {X 0,Y 740.072,Z 691.832,A -85,B 0,C 180,E1 1868.888,E2 1868.888} C_VEL
LIN {X 0,Y 739.609,Z 728.027,A -85,B 0,C 180,E1 1870.617,E2 1870.617} C_VEL
LIN {X 0,Y 739.156,Z 760.624,A -85,B 0,C 180,E1 1872.708,E2 1872.708} C_VEL
LIN {X 0,Y 738.814,Z 789.494,A -85,B 0,C 180,E1 1875.143,E2 1875.143} C_VEL
LIN {X 0,Y 738.589,Z 813.887,A -85,B 0,C 180,E1 1877.858,E2 1877.858} C_VEL
LIN {X 0,Y 738.405,Z 833.468,A -85,B 0,C 180,E1 1880.846,E2 1880.846} C_VEL
LIN {X 0,Y 738.34,Z 846.777,A -85,B 0,C 180,E1 1883.812,E2 1883.812} C_VEL
LIN {X 0,Y 738.334,Z 854.02,A -85,B 0,C 180,E1 1886.467,E2 1886.467} C_VEL
LIN {X 0,Y 738.289,Z 857.11,A -85,B 0,C 180,E1 1888.821,E2 1888.821} C_VEL
LIN {X 0,Y 738.334,Z 857.045,A -85,B 0,C 180,E1 1891.173,E2 1891.173} C_VEL
LIN {X 0,Y 738.388,Z 852.604,A -85,B 0,C 180,E1 1894.115,E2 1894.115} C_VEL
LIN {X 0,Y 738.412,Z 843.024,A -85,B 0,C 180,E1 1897.069,E2 1897.069} C_VEL
LIN {X 0,Y 738.552,Z 827.478,A -85,B 0,C 180,E1 1900.093,E2 1900.093} C_VEL
LIN {X 0,Y 738.691,Z 805.839,A -85,B 0,C 180,E1 1903.037,E2 1903.037} C_VEL
LIN {X 0,Y 738.984,Z 780.575,A -85,B 0,C 180,E1 1905.593,E2 1905.593} C_VEL
LIN {X 0,Y 739.306,Z 750.694,A -85,B 0,C 180,E1 1907.901,E2 1907.901} C_VEL
LIN {X 0,Y 739.737,Z 716.327,A -85,B 0,C 180,E1 1909.913,E2 1909.913} C_VEL
LIN {X 0,Y 740.16,Z 679.467,A -85,B 0,C 180,E1 1911.496,E2 1911.496} C_VEL
LIN {X 0,Y 740.527,Z 639.818,A -85,B 0,C 180,E1 1912.656,E2 1912.656} C_VEL
LIN {X 0,Y 739.84,Z 606.818,A -85,B 0,C 180,E1 1913.275,E2 1913.275} C_VEL
LIN {X 0,Y 738.283,Z 601.31,A -85,B 0,C 180,E1 1913.428,E2 1913.428} C_VEL
LIN {X 0,Y 737.939,Z 601.31,A -85,B 0,C 180,E1 1919.52,E2 1919.52} C_VEL
LIN {X 0,Y 737.959,Z 601.31,A -85,B 0,C 180,E1 1923.664,E2 1923.664} C_VEL
LIN {X 0,Y 737.842,Z 601.31,A -85,B 0,C 180,E1 1928.725,E2 1928.725} C_VEL
LIN {X 0,Y 738.207,Z 601.31,A -85,B 0,C 180,E1 1934.251,E2 1934.251} C_VEL
LIN {X 0,Y 738.011,Z 601.31,A -85,B 0,C 180,E1 1940.484,E2 1940.484} C_VEL
LIN {X 0,Y 737.973,Z 601.31,A -85,B 0,C 180,E1 1945.207,E2 1945.207} C_VEL
LIN {X 0,Y 737.917,Z 601.31,A -85,B 0,C 180,E1 1950.484,E2 1950.484} C_VEL
LIN {X 0,Y 738.131,Z 601.31,A -85,B 0,C 180,E1 1954.576,E2 1954.576} C_VEL
LIN {X 0,Y 738.019,Z 601.31,A -85,B 0,C 180,E1 1958.318,E2 1958.318} C_VEL
LIN {X 0,Y 738.211,Z 601.31,A -85,B 0,C 180,E1 1962.602,E2 1962.602} C_VEL
LIN {X 0,Y 739.669,Z 621.778,A -85,B 0,C 180,E1 1962.863,E2 1962.863} C_VEL
LIN {X 0,Y 739.64,Z 690.848,A -85,B 0,C 180,E1 1963.632,E2 1963.632} C_VEL
LIN {X 0,Y 739.456,Z 724.253,A -85,B 0,C 180,E1 1964.466,E2 1964.466} C_VEL
LIN {X 0,Y 739.171,Z 756.381,A -85,B 0,C 180,E1 1965.765,E2 1965.765} C_VEL
LIN {X 0,Y 738.888,Z 785.707,A -85,B 0,C 180,E1 1967.495,E2 1967.495} C_VEL
LIN {X 0,Y 738.699,Z 810.463,A -85,B 0,C 180,E1 1969.543,E2 1969.543} C_VEL
LIN {X 0,Y 738.531,Z 830.601,A -85,B 0,C 180,E1 1971.895,E2 1971.895} C_VEL
LIN {X 0,Y 738.463,Z 845.276,A -85,B 0,C 180,E1 1974.44,E2 1974.44} C_VEL
LIN {X 0,Y 738.375,Z 854.206,A -85,B 0,C 180,E1 1977.061,E2 1977.061} C_VEL
LIN {X 0,Y 738.363,Z 857.16,A -85,B 0,C 180,E1 1979.27,E2 1979.27} C_VEL
LIN {X 0,Y 738.369,Z 855.852,A -85,B 0,C 180,E1 1981.902,E2 1981.902} C_VEL
LIN {X 0,Y 737.153,Z 854.783,A -85,B 0,C 180,E1 1982.57,E2 1982.57} C_VEL
LIN {X 0,Y 730.674,Z 849.984,A -85,B 0,C 180,E1 1984.36,E2 1984.36} C_VEL
LIN {X 0,Y 730.565,Z 849.368,A -85,B 0,C 180,E1 1984.526,E2 1984.526} C_VEL
LIN {X 0,Y 730.632,Z 836.822,A -85,B 0,C 180,E1 1987.148,E2 1987.148} C_VEL
LIN {X 0,Y 730.757,Z 819.206,A -85,B 0,C 180,E1 1989.548,E2 1989.548} C_VEL
LIN {X 0,Y 730.967,Z 797.409,A -85,B 0,C 180,E1 1991.659,E2 1991.659} C_VEL
LIN {X 0,Y 731.309,Z 770.166,A -85,B 0,C 180,E1 1993.554,E2 1993.554} C_VEL
LIN {X 0,Y 731.675,Z 740.819,A -85,B 0,C 180,E1 1995.001,E2 1995.001} C_VEL
LIN {X 0,Y 731.98,Z 707.524,A -85,B 0,C 180,E1 1996.093,E2 1996.093} C_VEL
LIN {X 0,Y 732.066,Z 674.987,A -85,B 0,C 180,E1 1996.687,E2 1996.687} C_VEL
LIN {X 0,Y 731.408,Z 606.038,A -85,B 0,C 180,E1 1997.404,E2 1997.404} C_VEL
LIN {X 0,Y 730.34,Z 601.31,A -85,B 0,C 180,E1 1997.533,E2 1997.533} C_VEL
LIN {X 0,Y 730.031,Z 601.31,A -85,B 0,C 180,E1 2001.934,E2 2001.934} C_VEL
LIN {X 0,Y 730.031,Z 601.31,A -85,B 0,C 180,E1 2005.836,E2 2005.836} C_VEL
LIN {X 0,Y 730.022,Z 601.31,A -85,B 0,C 180,E1 2009.871,E2 2009.871} C_VEL
LIN {X 0,Y 729.988,Z 601.31,A -85,B 0,C 180,E1 2014.079,E2 2014.079} C_VEL
LIN {X 0,Y 730.039,Z 601.31,A -85,B 0,C 180,E1 2018.502,E2 2018.502} C_VEL
LIN {X 0,Y 730.209,Z 601.31,A -85,B 0,C 180,E1 2023.431,E2 2023.431} C_VEL
LIN {X 0,Y 729.866,Z 601.31,A -85,B 0,C 180,E1 2028.374,E2 2028.374} C_VEL
LIN {X 0,Y 729.888,Z 601.31,A -85,B 0,C 180,E1 2032.989,E2 2032.989} C_VEL
LIN {X 0,Y 729.961,Z 601.31,A -85,B 0,C 180,E1 2038.309,E2 2038.309} C_VEL
LIN {X 0,Y 730.108,Z 602.01,A -85,B 0,C 180,E1 2038.655,E2 2038.655} C_VEL
LIN {X 0,Y 734.226,Z 613.494,A -85,B 0,C 180,E1 2038.979,E2 2038.979} C_VEL
LIN {X 0,Y 735.345,Z 638.05,A -85,B 0,C 180,E1 2039.305,E2 2039.305} C_VEL
LIN {X 0,Y 735.115,Z 709.289,A -85,B 0,C 180,E1 2040.198,E2 2040.198} C_VEL
LIN {X 0,Y 734.453,Z 752.306,A -85,B 0,C 180,E1 2041.2,E2 2041.2} C_VEL
LIN {X 0,Y 733.837,Z 795.417,A -85,B 0,C 180,E1 2042.708,E2 2042.708} C_VEL
LIN {X 0,Y 733.015,Z 838.199,A -85,B 0,C 180,E1 2044.769,E2 2044.769} C_VEL
LIN {X 0,Y 732.209,Z 878.121,A -85,B 0,C 180,E1 2047.31,E2 2047.31} C_VEL
LIN {X 0,Y 731.521,Z 913.255,A -85,B 0,C 180,E1 2050.196,E2 2050.196} C_VEL
LIN {X 0,Y 730.924,Z 942.596,A -85,B 0,C 180,E1 2053.287,E2 2053.287} C_VEL
LIN {X 0,Y 730.637,Z 964.234,A -85,B 0,C 180,E1 2056.206,E2 2056.206} C_VEL
LIN {X 0,Y 730.497,Z 983.257,A -85,B 0,C 180,E1 2059.568,E2 2059.568} C_VEL
LIN {X 0,Y 730.4,Z 996.17,A -85,B 0,C 180,E1 2062.853,E2 2062.853} C_VEL
LIN {X 0,Y 730.429,Z 1003.669,A -85,B 0,C 180,E1 2065.84,E2 2065.84} C_VEL
LIN {X 0,Y 730.455,Z 1007.171,A -85,B 0,C 180,E1 2068.815,E2 2068.815} C_VEL
LIN {X 0,Y 730.521,Z 1006.218,A -85,B 0,C 180,E1 2072.381,E2 2072.381} C_VEL
LIN {X 0,Y 730.506,Z 999.626,A -85,B 0,C 180,E1 2075.956,E2 2075.956} C_VEL
LIN {X 0,Y 730.501,Z 988.507,A -85,B 0,C 180,E1 2079.254,E2 2079.254} C_VEL
LIN {X 0,Y 730.624,Z 970.984,A -85,B 0,C 180,E1 2082.716,E2 2082.716} C_VEL
LIN {X 0,Y 730.869,Z 948.738,A -85,B 0,C 180,E1 2085.947,E2 2085.947} C_VEL
LIN {X 0,Y 731.329,Z 921.054,A -85,B 0,C 180,E1 2089.049,E2 2089.049} C_VEL
LIN {X 0,Y 731.965,Z 888.848,A -85,B 0,C 180,E1 2091.88,E2 2091.88} C_VEL
LIN {X 0,Y 732.767,Z 851.909,A -85,B 0,C 180,E1 2094.432,E2 2094.432} C_VEL
LIN {X 0,Y 733.615,Z 810.585,A -85,B 0,C 180,E1 2096.627,E2 2096.627} C_VEL
LIN {X 0,Y 734.377,Z 768.287,A -85,B 0,C 180,E1 2098.295,E2 2098.295} C_VEL
LIN {X 0,Y 734.998,Z 726.748,A -85,B 0,C 180,E1 2099.449,E2 2099.449} C_VEL
LIN {X 0,Y 735.235,Z 685.128,A -85,B 0,C 180,E1 2100.167,E2 2100.167} C_VEL
LIN {X 0,Y 734.773,Z 612.92,A -85,B 0,C 180,E1 2101.001,E2 2101.001} C_VEL
LIN {X 0,Y 730.365,Z 601.31,A -85,B 0,C 180,E1 2101.376,E2 2101.376} C_VEL
LIN {X 0,Y 730.085,Z 601.31,A -85,B 0,C 180,E1 2107.007,E2 2107.007} C_VEL
LIN {X 0,Y 730.033,Z 601.31,A -85,B 0,C 180,E1 2111.664,E2 2111.664} C_VEL
LIN {X 0,Y 730.127,Z 601.31,A -85,B 0,C 180,E1 2115.133,E2 2115.133} C_VEL
LIN {X 0,Y 730.07,Z 601.31,A -85,B 0,C 180,E1 2120.171,E2 2120.171} C_VEL
LIN {X 0,Y 729.943,Z 601.31,A -85,B 0,C 180,E1 2124.471,E2 2124.471} C_VEL
LIN {X 0,Y 730.08,Z 601.31,A -85,B 0,C 180,E1 2128.751,E2 2128.751} C_VEL
LIN {X 0,Y 730.183,Z 601.31,A -85,B 0,C 180,E1 2134.17,E2 2134.17} C_VEL
LIN {X 0,Y 730.075,Z 601.31,A -85,B 0,C 180,E1 2139.066,E2 2139.066} C_VEL
LIN {X 0,Y 730.179,Z 601.31,A -85,B 0,C 180,E1 2143.113,E2 2143.113} C_VEL
LIN {X 0,Y 730.014,Z 601.31,A -85,B 0,C 180,E1 2148.022,E2 2148.022} C_VEL
LIN {X 0,Y 730.321,Z 601.31,A -85,B 0,C 180,E1 2152.849,E2 2152.849} C_VEL
LIN {X 0,Y 730.361,Z 601.31,A -85,B 0,C 180,E1 2157.621,E2 2157.621} C_VEL
LIN {X 0,Y 730.213,Z 601.31,A -85,B 0,C 180,E1 2162.376,E2 2162.376} C_VEL
LIN {X 0,Y 730.197,Z 601.31,A -85,B 0,C 180,E1 2165.953,E2 2165.953} C_VEL
LIN {X 0,Y 730.145,Z 601.31,A -85,B 0,C 180,E1 2170.76,E2 2170.76} C_VEL
LIN {X 0,Y 730.232,Z 601.31,A -85,B 0,C 180,E1 2175.644,E2 2175.644} C_VEL
LIN {X 0,Y 730.146,Z 601.31,A -85,B 0,C 180,E1 2180.949,E2 2180.949} C_VEL
LIN {X 0,Y 730.032,Z 601.31,A -85,B 0,C 180,E1 2185.833,E2 2185.833} C_VEL
LIN {X 0,Y 730.019,Z 601.31,A -85,B 0,C 180,E1 2189.868,E2 2189.868} C_VEL
LIN {X 0,Y 729.985,Z 601.31,A -85,B 0,C 180,E1 2194.075,E2 2194.075} C_VEL
LIN {X 0,Y 730.025,Z 601.31,A -85,B 0,C 180,E1 2198.499,E2 2198.499} C_VEL
LIN {X 0,Y 730.191,Z 601.31,A -85,B 0,C 180,E1 2203.42,E2 2203.42} C_VEL
LIN {X 0,Y 729.893,Z 601.31,A -85,B 0,C 180,E1 2208.367,E2 2208.367} C_VEL
LIN {X 0,Y 729.92,Z 601.31,A -85,B 0,C 180,E1 2212.983,E2 2212.983} C_VEL
LIN {X 0,Y 730.047,Z 601.31,A -85,B 0,C 180,E1 2218.293,E2 2218.293} C_VEL
LIN {X 0,Y 730.248,Z 601.31,A -85,B 0,C 180,E1 2223.125,E2 2223.125} C_VEL
LIN {X 0,Y 730.311,Z 601.31,A -85,B 0,C 180,E1 2226.219,E2 2226.219} C_VEL
LIN {X 0,Y 733.25,Z 613.643,A -85,B 0,C 180,E1 2226.508,E2 2226.508} C_VEL
LIN {X 0,Y 733.111,Z 653.519,A -85,B 0,C 180,E1 2227.364,E2 2227.364} C_VEL
LIN {X 0,Y 732.59,Z 691.881,A -85,B 0,C 180,E1 2228.664,E2 2228.664} C_VEL
LIN {X 0,Y 732.056,Z 728.026,A -85,B 0,C 180,E1 2230.408,E2 2230.408} C_VEL
LIN {X 0,Y 731.475,Z 761.029,A -85,B 0,C 180,E1 2232.552,E2 2232.552} C_VEL
LIN {X 0,Y 731.072,Z 789.79,A -85,B 0,C 180,E1 2235.011,E2 2235.011} C_VEL
LIN {X 0,Y 730.75,Z 814.148,A -85,B 0,C 180,E1 2237.762,E2 2237.762} C_VEL
LIN {X 0,Y 730.533,Z 833.459,A -85,B 0,C 180,E1 2240.747,E2 2240.747} C_VEL
LIN {X 0,Y 730.46,Z 846.776,A -85,B 0,C 180,E1 2243.745,E2 2243.745} C_VEL
LIN {X 0,Y 730.435,Z 854.022,A -85,B 0,C 180,E1 2246.429,E2 2246.429} C_VEL
LIN {X 0,Y 730.389,Z 857.105,A -85,B 0,C 180,E1 2248.808,E2 2248.808} C_VEL
LIN {X 0,Y 730.433,Z 857.042,A -85,B 0,C 180,E1 2251.185,E2 2251.185} C_VEL
LIN {X 0,Y 730.522,Z 852.599,A -85,B 0,C 180,E1 2254.16,E2 2254.16} C_VEL
LIN {X 0,Y 730.581,Z 841.752,A -85,B 0,C 180,E1 2257.445,E2 2257.445} C_VEL
LIN {X 0,Y 730.658,Z 825.715,A -85,B 0,C 180,E1 2260.478,E2 2260.478} C_VEL
LIN {X 0,Y 730.908,Z 804.512,A -85,B 0,C 180,E1 2263.331,E2 2263.331} C_VEL
LIN {X 0,Y 731.271,Z 778.65,A -85,B 0,C 180,E1 2265.931,E2 2265.931} C_VEL
LIN {X 0,Y 731.759,Z 747.258,A -85,B 0,C 180,E1 2268.326,E2 2268.326} C_VEL
LIN {X 0,Y 732.317,Z 712.078,A -85,B 0,C 180,E1 2270.343,E2 2270.343} C_VEL
LIN {X 0,Y 732.854,Z 673.958,A -85,B 0,C 180,E1 2271.917,E2 2271.917} C_VEL
LIN {X 0,Y 733.329,Z 634.171,A -85,B 0,C 180,E1 2273.021,E2 2273.021} C_VEL
LIN {X 0,Y 732.654,Z 608.703,A -85,B 0,C 180,E1 2273.492,E2 2273.492} C_VEL
LIN {X 0,Y 730.277,Z 601.31,A -85,B 0,C 180,E1 2273.706,E2 2273.706} C_VEL
LIN {X 0,Y 730.027,Z 601.31,A -85,B 0,C 180,E1 2279.365,E2 2279.365} C_VEL
LIN {X 0,Y 729.989,Z 601.31,A -85,B 0,C 180,E1 2284.081,E2 2284.081} C_VEL
LIN {X 0,Y 729.969,Z 601.31,A -85,B 0,C 180,E1 2288.51,E2 2288.51} C_VEL
LIN {X 0,Y 730.203,Z 601.31,A -85,B 0,C 180,E1 2293.441,E2 2293.441} C_VEL
LIN {X 0,Y 729.906,Z 601.31,A -85,B 0,C 180,E1 2298.385,E2 2298.385} C_VEL
LIN {X 0,Y 729.912,Z 601.31,A -85,B 0,C 180,E1 2302.998,E2 2302.998} C_VEL
LIN {X 0,Y 730.049,Z 601.31,A -85,B 0,C 180,E1 2308.309,E2 2308.309} C_VEL
LIN {X 0,Y 730.246,Z 601.31,A -85,B 0,C 180,E1 2313.146,E2 2313.146} C_VEL
LIN {X 0,Y 730.155,Z 601.31,A -85,B 0,C 180,E1 2318.073,E2 2318.073} C_VEL
LIN {X 0,Y 730.237,Z 601.31,A -85,B 0,C 180,E1 2322.406,E2 2322.406} C_VEL
LIN {X 0,Y 732.126,Z 619.293,A -85,B 0,C 180,E1 2322.657,E2 2322.657} C_VEL
LIN {X 0,Y 732.053,Z 691.472,A -85,B 0,C 180,E1 2323.47,E2 2323.47} C_VEL
LIN {X 0,Y 731.812,Z 725.664,A -85,B 0,C 180,E1 2324.345,E2 2324.345} C_VEL
LIN {X 0,Y 731.484,Z 756.371,A -85,B 0,C 180,E1 2325.612,E2 2325.612} C_VEL
LIN {X 0,Y 731.141,Z 785.007,A -85,B 0,C 180,E1 2327.31,E2 2327.31} C_VEL
LIN {X 0,Y 730.872,Z 810.101,A -85,B 0,C 180,E1 2329.394,E2 2329.394} C_VEL
LIN {X 0,Y 730.655,Z 829.511,A -85,B 0,C 180,E1 2331.657,E2 2331.657} C_VEL
LIN {X 0,Y 730.603,Z 843.799,A -85,B 0,C 180,E1 2334.051,E2 2334.051} C_VEL
LIN {X 0,Y 730.567,Z 852.689,A -85,B 0,C 180,E1 2336.435,E2 2336.435} C_VEL
LIN {X 0,Y 730.503,Z 856.957,A -85,B 0,C 180,E1 2338.813,E2 2338.813} C_VEL
LIN {X 0,Y 730.526,Z 856.878,A -85,B 0,C 180,E1 2341.19,E2 2341.19} C_VEL
LIN {X 0,Y 730.593,Z 852.444,A -85,B 0,C 180,E1 2343.568,E2 2343.568} C_VEL
LIN {X 0,Y 730.565,Z 849.368,A -85,B 0,C 180,E1 2344.526,E2 2344.526} C_VEL
LIN {X 0,Y 726.625,Z 844.187,A -85,B 0,C 180,E1 2345.805,E2 2345.805} C_VEL
LIN {X 0,Y 722.746,Z 837.754,A -85,B 0,C 180,E1 2347.065,E2 2347.065} C_VEL
LIN {X 0,Y 722.9,Z 820.536,A -85,B 0,C 180,E1 2349.5,E2 2349.5} C_VEL
LIN {X 0,Y 723.175,Z 797.415,A -85,B 0,C 180,E1 2351.787,E2 2351.787} C_VEL
LIN {X 0,Y 723.588,Z 770.171,A -85,B 0,C 180,E1 2353.701,E2 2353.701} C_VEL
LIN {X 0,Y 724.025,Z 739.733,A -85,B 0,C 180,E1 2355.208,E2 2355.208} C_VEL
LIN {X 0,Y 724.371,Z 706.835,A -85,B 0,C 180,E1 2356.284,E2 2356.284} C_VEL
LIN {X 0,Y 724.56,Z 671.785,A -85,B 0,C 180,E1 2356.904,E2 2356.904} C_VEL
LIN {X 0,Y 723.714,Z 606.686,A -85,B 0,C 180,E1 2357.589,E2 2357.589} C_VEL
LIN {X 0,Y 722.395,Z 601.31,A -85,B 0,C 180,E1 2357.743,E2 2357.743} C_VEL
LIN {X 0,Y 722.117,Z 601.31,A -85,B 0,C 180,E1 2362.604,E2 2362.604} C_VEL
LIN {X 0,Y 722.147,Z 601.31,A -85,B 0,C 180,E1 2367.486,E2 2367.486} C_VEL
LIN {X 0,Y 722.166,Z 601.31,A -85,B 0,C 180,E1 2373.054,E2 2373.054} C_VEL
LIN {X 0,Y 722.249,Z 601.31,A -85,B 0,C 180,E1 2377.466,E2 2377.466} C_VEL
LIN {X 0,Y 722.223,Z 601.31,A -85,B 0,C 180,E1 2382.758,E2 2382.758} C_VEL
LIN {X 0,Y 721.956,Z 601.31,A -85,B 0,C 180,E1 2387.259,E2 2387.259} C_VEL
LIN {X 0,Y 721.994,Z 601.31,A -85,B 0,C 180,E1 2392.515,E2 2392.515} C_VEL
LIN {X 0,Y 721.946,Z 601.31,A -85,B 0,C 180,E1 2397.072,E2 2397.072} C_VEL
LIN {X 0,Y 722.101,Z 601.984,A -85,B 0,C 180,E1 2398.267,E2 2398.267} C_VEL
LIN {X 0,Y 727.694,Z 616.774,A -85,B 0,C 180,E1 2398.707,E2 2398.707} C_VEL
LIN {X 0,Y 728.511,Z 651.806,A -85,B 0,C 180,E1 2399.141,E2 2399.141} C_VEL
LIN {X 0,Y 728.155,Z 713.738,A -85,B 0,C 180,E1 2399.963,E2 2399.963} C_VEL
LIN {X 0,Y 727.352,Z 760.318,A -85,B 0,C 180,E1 2401.137,E2 2401.137} C_VEL
LIN {X 0,Y 726.465,Z 803.579,A -85,B 0,C 180,E1 2402.771,E2 2402.771} C_VEL
LIN {X 0,Y 725.577,Z 842.382,A -85,B 0,C 180,E1 2404.74,E2 2404.74} C_VEL
LIN {X 0,Y 724.643,Z 880.073,A -85,B 0,C 180,E1 2407.209,E2 2407.209} C_VEL
LIN {X 0,Y 723.821,Z 914.689,A -85,B 0,C 180,E1 2410.117,E2 2410.117} C_VEL
LIN {X 0,Y 723.156,Z 943.918,A -85,B 0,C 180,E1 2413.259,E2 2413.259} C_VEL
LIN {X 0,Y 722.745,Z 968.166,A -85,B 0,C 180,E1 2416.67,E2 2416.67} C_VEL
LIN {X 0,Y 722.618,Z 985.695,A -85,B 0,C 180,E1 2420.006,E2 2420.006} C_VEL
LIN {X 0,Y 722.517,Z 998.079,A -85,B 0,C 180,E1 2423.38,E2 2423.38} C_VEL
LIN {X 0,Y 722.451,Z 1004.657,A -85,B 0,C 180,E1 2426.396,E2 2426.396} C_VEL
LIN {X 0,Y 722.473,Z 1007.5,A -85,B 0,C 180,E1 2430.003,E2 2430.003} C_VEL
LIN {X 0,Y 722.507,Z 1004.648,A -85,B 0,C 180,E1 2433.61,E2 2433.61} C_VEL
LIN {X 0,Y 722.511,Z 998.06,A -85,B 0,C 180,E1 2436.627,E2 2436.627} C_VEL
LIN {X 0,Y 722.632,Z 985.8,A -85,B 0,C 180,E1 2439.97,E2 2439.97} C_VEL
LIN {X 0,Y 722.785,Z 969.552,A -85,B 0,C 180,E1 2443.108,E2 2443.108} C_VEL
LIN {X 0,Y 723.095,Z 946.309,A -85,B 0,C 180,E1 2446.436,E2 2446.436} C_VEL
LIN {X 0,Y 723.622,Z 919.444,A -85,B 0,C 180,E1 2449.419,E2 2449.419} C_VEL
LIN {X 0,Y 724.436,Z 887.221,A -85,B 0,C 180,E1 2452.245,E2 2452.245} C_VEL
LIN {X 0,Y 725.389,Z 850.07,A -85,B 0,C 180,E1 2454.807,E2 2454.807} C_VEL
LIN {X 0,Y 726.459,Z 808.908,A -85,B 0,C 180,E1 2456.992,E2 2456.992} C_VEL
LIN {X 0,Y 727.363,Z 767.167,A -85,B 0,C 180,E1 2458.632,E2 2458.632} C_VEL
LIN {X 0,Y 728.123,Z 726.511,A -85,B 0,C 180,E1 2459.76,E2 2459.76} C_VEL
LIN {X 0,Y 728.414,Z 683.558,A -85,B 0,C 180,E1 2460.5,E2 2460.5} C_VEL
LIN {X 0,Y 728.012,Z 614.963,A -85,B 0,C 180,E1 2461.299,E2 2461.299} C_VEL
LIN {X 0,Y 722.435,Z 601.31,A -85,B 0,C 180,E1 2461.752,E2 2461.752} C_VEL
LIN {X 0,Y 722.157,Z 601.31,A -85,B 0,C 180,E1 2467.483,E2 2467.483} C_VEL
LIN {X 0,Y 722.203,Z 601.31,A -85,B 0,C 180,E1 2472.762,E2 2472.762} C_VEL
LIN {X 0,Y 721.944,Z 601.31,A -85,B 0,C 180,E1 2477.818,E2 2477.818} C_VEL
LIN {X 0,Y 722.041,Z 601.31,A -85,B 0,C 180,E1 2482.891,E2 2482.891} C_VEL
LIN {X 0,Y 722.143,Z 601.31,A -85,B 0,C 180,E1 2488.368,E2 2488.368} C_VEL
LIN {X 0,Y 722.27,Z 601.31,A -85,B 0,C 180,E1 2493.866,E2 2493.866} C_VEL
LIN {X 0,Y 722.293,Z 601.31,A -85,B 0,C 180,E1 2497.818,E2 2497.818} C_VEL
LIN {X 0,Y 722.287,Z 601.31,A -85,B 0,C 180,E1 2502.923,E2 2502.923} C_VEL
LIN {X 0,Y 722.109,Z 601.31,A -85,B 0,C 180,E1 2507.889,E2 2507.889} C_VEL
LIN {X 0,Y 722.397,Z 601.31,A -85,B 0,C 180,E1 2512.77,E2 2512.77} C_VEL
LIN {X 0,Y 722.456,Z 601.31,A -85,B 0,C 180,E1 2517.595,E2 2517.595} C_VEL
LIN {X 0,Y 722.311,Z 601.31,A -85,B 0,C 180,E1 2522.402,E2 2522.402} C_VEL
LIN {X 0,Y 722.287,Z 601.31,A -85,B 0,C 180,E1 2526.018,E2 2526.018} C_VEL
LIN {X 0,Y 722.242,Z 601.31,A -85,B 0,C 180,E1 2530.88,E2 2530.88} C_VEL
LIN {X 0,Y 722.345,Z 601.31,A -85,B 0,C 180,E1 2535.819,E2 2535.819} C_VEL
LIN {X 0,Y 722.282,Z 601.31,A -85,B 0,C 180,E1 2540.887,E2 2540.887} C_VEL
LIN {X 0,Y 722.16,Z 601.31,A -85,B 0,C 180,E1 2545.543,E2 2545.543} C_VEL
LIN {X 0,Y 722.09,Z 601.31,A -85,B 0,C 180,E1 2550.64,E2 2550.64} C_VEL
LIN {X 0,Y 722.055,Z 601.31,A -85,B 0,C 180,E1 2555.069,E2 2555.069} C_VEL
LIN {X 0,Y 722.032,Z 601.31,A -85,B 0,C 180,E1 2559.058,E2 2559.058} C_VEL
LIN {X 0,Y 722.247,Z 601.31,A -85,B 0,C 180,E1 2564.492,E2 2564.492} C_VEL
LIN {X 0,Y 722.057,Z 601.31,A -85,B 0,C 180,E1 2569.415,E2 2569.415} C_VEL
LIN {X 0,Y 722.04,Z 601.31,A -85,B 0,C 180,E1 2574.907,E2 2574.907} C_VEL
LIN {X 0,Y 722.131,Z 601.31,A -85,B 0,C 180,E1 2579.759,E2 2579.759} C_VEL
LIN {X 0,Y 722.328,Z 601.31,A -85,B 0,C 180,E1 2585.191,E2 2585.191} C_VEL
LIN {X 0,Y 722.388,Z 601.31,A -85,B 0,C 180,E1 2585.951,E2 2585.951} C_VEL
LIN {X 0,Y 726.01,Z 614.737,A -85,B 0,C 180,E1 2586.277,E2 2586.277} C_VEL
LIN {X 0,Y 725.775,Z 654.845,A -85,B 0,C 180,E1 2587.162,E2 2587.162} C_VEL
LIN {X 0,Y 725.137,Z 692.984,A -85,B 0,C 180,E1 2588.481,E2 2588.481} C_VEL
LIN {X 0,Y 724.485,Z 729.253,A -85,B 0,C 180,E1 2590.266,E2 2590.266} C_VEL
LIN {X 0,Y 723.776,Z 762.664,A -85,B 0,C 180,E1 2592.485,E2 2592.485} C_VEL
LIN {X 0,Y 723.223,Z 791.957,A -85,B 0,C 180,E1 2595.059,E2 2595.059} C_VEL
LIN {X 0,Y 722.885,Z 816.099,A -85,B 0,C 180,E1 2597.897,E2 2597.897} C_VEL
LIN {X 0,Y 722.673,Z 833.449,A -85,B 0,C 180,E1 2600.645,E2 2600.645} C_VEL
LIN {X 0,Y 722.559,Z 846.773,A -85,B 0,C 180,E1 2603.676,E2 2603.676} C_VEL
LIN {X 0,Y 722.539,Z 854.025,A -85,B 0,C 180,E1 2606.39,E2 2606.39} C_VEL
LIN {X 0,Y 722.49,Z 857.1,A -85,B 0,C 180,E1 2608.795,E2 2608.795} C_VEL
LIN {X 0,Y 722.562,Z 857.038,A -85,B 0,C 180,E1 2611.198,E2 2611.198} C_VEL
LIN {X 0,Y 722.641,Z 852.594,A -85,B 0,C 180,E1 2614.205,E2 2614.205} C_VEL
LIN {X 0,Y 722.699,Z 841.756,A -85,B 0,C 180,E1 2617.526,E2 2617.526} C_VEL
LIN {X 0,Y 722.794,Z 825.679,A -85,B 0,C 180,E1 2620.599,E2 2620.599} C_VEL
LIN {X 0,Y 723.095,Z 804.521,A -85,B 0,C 180,E1 2623.477,E2 2623.477} C_VEL
LIN {X 0,Y 723.545,Z 778.66,A -85,B 0,C 180,E1 2626.106,E2 2626.106} C_VEL
LIN {X 0,Y 724.109,Z 748.414,A -85,B 0,C 180,E1 2628.447,E2 2628.447} C_VEL
LIN {X 0,Y 724.744,Z 714.306,A -85,B 0,C 180,E1 2630.45,E2 2630.45} C_VEL
LIN {X 0,Y 725.43,Z 677.333,A -85,B 0,C 180,E1 2632.035,E2 2632.035} C_VEL
LIN {X 0,Y 726.026,Z 636.368,A -85,B 0,C 180,E1 2633.216,E2 2633.216} C_VEL
LIN {X 0,Y 725.404,Z 610.841,A -85,B 0,C 180,E1 2633.713,E2 2633.713} C_VEL
LIN {X 0,Y 722.287,Z 601.31,A -85,B 0,C 180,E1 2634.025,E2 2634.025} C_VEL
LIN {X 0,Y 722.137,Z 601.31,A -85,B 0,C 180,E1 2638.851,E2 2638.851} C_VEL
LIN {X 0,Y 722.168,Z 601.31,A -85,B 0,C 180,E1 2643.056,E2 2643.056} C_VEL
LIN {X 0,Y 722.185,Z 601.31,A -85,B 0,C 180,E1 2647.473,E2 2647.473} C_VEL
LIN {X 0,Y 722.209,Z 601.31,A -85,B 0,C 180,E1 2652.767,E2 2652.767} C_VEL
LIN {X 0,Y 721.974,Z 601.31,A -85,B 0,C 180,E1 2657.824,E2 2657.824} C_VEL
LIN {X 0,Y 722.02,Z 601.31,A -85,B 0,C 180,E1 2662.882,E2 2662.882} C_VEL
LIN {X 0,Y 722.181,Z 601.31,A -85,B 0,C 180,E1 2668.373,E2 2668.373} C_VEL
LIN {X 0,Y 722.312,Z 601.31,A -85,B 0,C 180,E1 2673.871,E2 2673.871} C_VEL
LIN {X 0,Y 722.235,Z 601.31,A -85,B 0,C 180,E1 2677.82,E2 2677.82} C_VEL
LIN {X 0,Y 722.249,Z 601.31,A -85,B 0,C 180,E1 2682.221,E2 2682.221} C_VEL
LIN {X 0,Y 724.589,Z 616.25,A -85,B 0,C 180,E1 2682.44,E2 2682.44} C_VEL
LIN {X 0,Y 724.467,Z 691.446,A -85,B 0,C 180,E1 2683.292,E2 2683.292} C_VEL
LIN {X 0,Y 724.215,Z 724.656,A -85,B 0,C 180,E1 2684.145,E2 2684.145} C_VEL
LIN {X 0,Y 723.808,Z 756.357,A -85,B 0,C 180,E1 2685.456,E2 2685.456} C_VEL
LIN {X 0,Y 723.4,Z 784.454,A -85,B 0,C 180,E1 2687.132,E2 2687.132} C_VEL
LIN {X 0,Y 723.051,Z 810.018,A -85,B 0,C 180,E1 2689.27,E2 2689.27} C_VEL
LIN {X 0,Y 722.798,Z 829.507,A -85,B 0,C 180,E1 2691.565,E2 2691.565} C_VEL
LIN {X 0,Y 722.694,Z 844.858,A -85,B 0,C 180,E1 2694.224,E2 2694.224} C_VEL
LIN {X 0,Y 722.671,Z 852.687,A -85,B 0,C 180,E1 2696.396,E2 2696.396} C_VEL
LIN {X 0,Y 722.603,Z 856.958,A -85,B 0,C 180,E1 2698.8,E2 2698.8} C_VEL
LIN {X 0,Y 722.624,Z 856.878,A -85,B 0,C 180,E1 2701.203,E2 2701.203} C_VEL
LIN {X 0,Y 722.693,Z 852.445,A -85,B 0,C 180,E1 2703.607,E2 2703.607} C_VEL
LIN {X 0,Y 722.73,Z 841.807,A -85,B 0,C 180,E1 2706.319,E2 2706.319} C_VEL
LIN {X 0,Y 722.746,Z 837.754,A -85,B 0,C 180,E1 2707.065,E2 2707.065} C_VEL
LIN {X 0,Y 718.857,Z 830.341,A -85,B 0,C 180,E1 2708.292,E2 2708.292} C_VEL
LIN {X 0,Y 715.033,Z 821.643,A -85,B 0,C 180,E1 2709.475,E2 2709.475} C_VEL
LIN {X 0,Y 715.354,Z 799.188,A -85,B 0,C 180,E1 2711.762,E2 2711.762} C_VEL
LIN {X 0,Y 715.829,Z 772.704,A -85,B 0,C 180,E1 2713.697,E2 2713.697} C_VEL
LIN {X 0,Y 716.295,Z 743.008,A -85,B 0,C 180,E1 2715.241,E2 2715.241} C_VEL
LIN {X 0,Y 716.766,Z 709.848,A -85,B 0,C 180,E1 2716.382,E2 2716.382} C_VEL
LIN {X 0,Y 716.972,Z 675.072,A -85,B 0,C 180,E1 2717.049,E2 2717.049} C_VEL
LIN {X 0,Y 716.386,Z 608.921,A -85,B 0,C 180,E1 2717.753,E2 2717.753} C_VEL
LIN {X 0,Y 714.501,Z 601.31,A -85,B 0,C 180,E1 2717.918,E2 2717.918} C_VEL
LIN {X 0,Y 714.218,Z 601.31,A -85,B 0,C 180,E1 2722.446,E2 2722.446} C_VEL
LIN {X 0,Y 714.195,Z 601.31,A -85,B 0,C 180,E1 2727.002,E2 2727.002} C_VEL
LIN {X 0,Y 714.284,Z 601.31,A -85,B 0,C 180,E1 2732.021,E2 2732.021} C_VEL
LIN {X 0,Y 714.284,Z 601.31,A -85,B 0,C 180,E1 2736.432,E2 2736.432} C_VEL
LIN {X 0,Y 714.237,Z 601.31,A -85,B 0,C 180,E1 2742.06,E2 2742.06} C_VEL
LIN {X 0,Y 714.18,Z 601.31,A -85,B 0,C 180,E1 2746.155,E2 2746.155} C_VEL
LIN {X 0,Y 714.076,Z 601.31,A -85,B 0,C 180,E1 2751.717,E2 2751.717} C_VEL
LIN {X 0,Y 714.011,Z 601.31,A -85,B 0,C 180,E1 2756.517,E2 2756.517} C_VEL
LIN {X 0,Y 714.094,Z 601.31,A -85,B 0,C 180,E1 2757.841,E2 2757.841} C_VEL
LIN {X 0,Y 721.038,Z 618.528,A -85,B 0,C 180,E1 2758.405,E2 2758.405} C_VEL
LIN {X 0,Y 721.693,Z 675.855,A -85,B 0,C 180,E1 2759.09,E2 2759.09} C_VEL
LIN {X 0,Y 721.045,Z 723.189,A -85,B 0,C 180,E1 2759.844,E2 2759.844} C_VEL
LIN {X 0,Y 720.303,Z 766.214,A -85,B 0,C 180,E1 2761.027,E2 2761.027} C_VEL
LIN {X 0,Y 719.233,Z 809.278,A -85,B 0,C 180,E1 2762.732,E2 2762.732} C_VEL
LIN {X 0,Y 717.987,Z 852.027,A -85,B 0,C 180,E1 2765.038,E2 2765.038} C_VEL
LIN {X 0,Y 716.826,Z 890.466,A -85,B 0,C 180,E1 2767.76,E2 2767.76} C_VEL
LIN {X 0,Y 715.914,Z 924.608,A -85,B 0,C 180,E1 2770.885,E2 2770.885} C_VEL
LIN {X 0,Y 715.291,Z 952.892,A -85,B 0,C 180,E1 2774.238,E2 2774.238} C_VEL
LIN {X 0,Y 714.867,Z 975.306,A -85,B 0,C 180,E1 2777.766,E2 2777.766} C_VEL
LIN {X 0,Y 714.781,Z 990.879,A -85,B 0,C 180,E1 2781.163,E2 2781.163} C_VEL
LIN {X 0,Y 714.678,Z 1001.205,A -85,B 0,C 180,E1 2784.529,E2 2784.529} C_VEL
LIN {X 0,Y 714.605,Z 1006.223,A -85,B 0,C 180,E1 2787.573,E2 2787.573} C_VEL
LIN {X 0,Y 714.576,Z 1007.169,A -85,B 0,C 180,E1 2791.218,E2 2791.218} C_VEL
LIN {X 0,Y 714.687,Z 1002.278,A -85,B 0,C 180,E1 2794.958,E2 2794.958} C_VEL
LIN {X 0,Y 714.663,Z 993.155,A -85,B 0,C 180,E1 2798.231,E2 2798.231} C_VEL
LIN {X 0,Y 714.927,Z 976.967,A -85,B 0,C 180,E1 2801.929,E2 2801.929} C_VEL
LIN {X 0,Y 715.322,Z 954.326,A -85,B 0,C 180,E1 2805.558,E2 2805.558} C_VEL
LIN {X 0,Y 715.859,Z 927.365,A -85,B 0,C 180,E1 2808.816,E2 2808.816} C_VEL
LIN {X 0,Y 716.664,Z 897.414,A -85,B 0,C 180,E1 2811.656,E2 2811.656} C_VEL
LIN {X 0,Y 717.665,Z 862.89,A -85,B 0,C 180,E1 2814.257,E2 2814.257} C_VEL
LIN {X 0,Y 718.836,Z 822.921,A -85,B 0,C 180,E1 2816.602,E2 2816.602} C_VEL
LIN {X 0,Y 720.043,Z 779.699,A -85,B 0,C 180,E1 2818.498,E2 2818.498} C_VEL
LIN {X 0,Y 720.975,Z 735.702,A -85,B 0,C 180,E1 2819.857,E2 2819.857} C_VEL
LIN {X 0,Y 721.507,Z 692.651,A -85,B 0,C 180,E1 2820.701,E2 2820.701} C_VEL
LIN {X 0,Y 721.273,Z 617.615,A -85,B 0,C 180,E1 2821.594,E2 2821.594} C_VEL
LIN {X 0,Y 714.449,Z 601.31,A -85,B 0,C 180,E1 2822.19,E2 2822.19} C_VEL
LIN {X 0,Y 714.147,Z 601.31,A -85,B 0,C 180,E1 2827.977,E2 2827.977} C_VEL
LIN {X 0,Y 714.353,Z 601.31,A -85,B 0,C 180,E1 2833.859,E2 2833.859} C_VEL
LIN {X 0,Y 714.076,Z 601.31,A -85,B 0,C 180,E1 2838.877,E2 2838.877} C_VEL
LIN {X 0,Y 714.122,Z 601.31,A -85,B 0,C 180,E1 2843.739,E2 2843.739} C_VEL
LIN {X 0,Y 714.242,Z 601.31,A -85,B 0,C 180,E1 2849.399,E2 2849.399} C_VEL
LIN {X 0,Y 714.308,Z 601.31,A -85,B 0,C 180,E1 2854.901,E2 2854.901} C_VEL
LIN {X 0,Y 714.287,Z 601.31,A -85,B 0,C 180,E1 2858.975,E2 2858.975} C_VEL
LIN {X 0,Y 714.309,Z 601.31,A -85,B 0,C 180,E1 2863.995,E2 2863.995} C_VEL
LIN {X 0,Y 714.406,Z 601.31,A -85,B 0,C 180,E1 2868.996,E2 2868.996} C_VEL
LIN {X 0,Y 714.508,Z 601.31,A -85,B 0,C 180,E1 2873.913,E2 2873.913} C_VEL
LIN {X 0,Y 714.413,Z 601.31,A -85,B 0,C 180,E1 2878.783,E2 2878.783} C_VEL
LIN {X 0,Y 714.41,Z 601.31,A -85,B 0,C 180,E1 2882.429,E2 2882.429} C_VEL
LIN {X 0,Y 714.386,Z 601.31,A -85,B 0,C 180,E1 2886.085,E2 2886.085} C_VEL
LIN {X 0,Y 714.336,Z 601.31,A -85,B 0,C 180,E1 2891.002,E2 2891.002} C_VEL
LIN {X 0,Y 714.421,Z 601.31,A -85,B 0,C 180,E1 2896,E2 2896} C_VEL
LIN {X 0,Y 714.364,Z 601.31,A -85,B 0,C 180,E1 2901.129,E2 2901.129} C_VEL
LIN {X 0,Y 714.284,Z 601.31,A -85,B 0,C 180,E1 2905.096,E2 2905.096} C_VEL
LIN {X 0,Y 714.177,Z 601.31,A -85,B 0,C 180,E1 2909.551,E2 2909.551} C_VEL
LIN {X 0,Y 714.138,Z 601.31,A -85,B 0,C 180,E1 2914.154,E2 2914.154} C_VEL
LIN {X 0,Y 714.175,Z 601.31,A -85,B 0,C 180,E1 2918.274,E2 2918.274} C_VEL
LIN {X 0,Y 714.363,Z 601.31,A -85,B 0,C 180,E1 2923.845,E2 2923.845} C_VEL
LIN {X 0,Y 714.101,Z 601.31,A -85,B 0,C 180,E1 2928.866,E2 2928.866} C_VEL
LIN {X 0,Y 714.151,Z 601.31,A -85,B 0,C 180,E1 2933.711,E2 2933.711} C_VEL
LIN {X 0,Y 714.248,Z 601.31,A -85,B 0,C 180,E1 2939.39,E2 2939.39} C_VEL
LIN {X 0,Y 714.419,Z 601.31,A -85,B 0,C 180,E1 2944.898,E2 2944.898} C_VEL
LIN {X 0,Y 714.495,Z 601.31,A -85,B 0,C 180,E1 2945.679,E2 2945.679} C_VEL
LIN {X 0,Y 718.779,Z 617.508,A -85,B 0,C 180,E1 2946.071,E2 2946.071} C_VEL
LIN {X 0,Y 718.435,Z 658.416,A -85,B 0,C 180,E1 2947.021,E2 2947.021} C_VEL
LIN {X 0,Y 717.697,Z 694.551,A -85,B 0,C 180,E1 2948.315,E2 2948.315} C_VEL
LIN {X 0,Y 716.925,Z 730.185,A -85,B 0,C 180,E1 2950.104,E2 2950.104} C_VEL
LIN {X 0,Y 716.078,Z 763.62,A -85,B 0,C 180,E1 2952.366,E2 2952.366} C_VEL
LIN {X 0,Y 715.472,Z 792.37,A -85,B 0,C 180,E1 2954.938,E2 2954.938} C_VEL
LIN {X 0,Y 715.056,Z 816.09,A -85,B 0,C 180,E1 2957.763,E2 2957.763} C_VEL
LIN {X 0,Y 714.771,Z 835.025,A -85,B 0,C 180,E1 2960.848,E2 2960.848} C_VEL
LIN {X 0,Y 714.68,Z 847.743,A -85,B 0,C 180,E1 2963.912,E2 2963.912} C_VEL
LIN {X 0,Y 714.641,Z 854.027,A -85,B 0,C 180,E1 2966.35,E2 2966.35} C_VEL
LIN {X 0,Y 714.591,Z 857.095,A -85,B 0,C 180,E1 2968.782,E2 2968.782} C_VEL
LIN {X 0,Y 714.66,Z 857.034,A -85,B 0,C 180,E1 2971.212,E2 2971.212} C_VEL
LIN {X 0,Y 714.76,Z 852.589,A -85,B 0,C 180,E1 2974.252,E2 2974.252} C_VEL
LIN {X 0,Y 714.781,Z 843.02,A -85,B 0,C 180,E1 2977.304,E2 2977.304} C_VEL
LIN {X 0,Y 714.923,Z 827.814,A -85,B 0,C 180,E1 2980.375,E2 2980.375} C_VEL
LIN {X 0,Y 715.283,Z 805.837,A -85,B 0,C 180,E1 2983.471,E2 2983.471} C_VEL
LIN {X 0,Y 715.78,Z 780.426,A -85,B 0,C 180,E1 2986.128,E2 2986.128} C_VEL
LIN {X 0,Y 716.453,Z 749.571,A -85,B 0,C 180,E1 2988.572,E2 2988.572} C_VEL
LIN {X 0,Y 717.241,Z 714.978,A -85,B 0,C 180,E1 2990.639,E2 2990.639} C_VEL
LIN {X 0,Y 718.044,Z 677.297,A -85,B 0,C 180,E1 2992.275,E2 2992.275} C_VEL
LIN {X 0,Y 718.725,Z 636.363,A -85,B 0,C 180,E1 2993.466,E2 2993.466} C_VEL
LIN {X 0,Y 718.212,Z 612.848,A -85,B 0,C 180,E1 2993.938,E2 2993.938} C_VEL
LIN {X 0,Y 714.304,Z 601.31,A -85,B 0,C 180,E1 2994.295,E2 2994.295} C_VEL
LIN {X 0,Y 714.17,Z 601.31,A -85,B 0,C 180,E1 2999.581,E2 2999.581} C_VEL
LIN {X 0,Y 714.132,Z 601.31,A -85,B 0,C 180,E1 3004.18,E2 3004.18} C_VEL
LIN {X 0,Y 714.136,Z 601.31,A -85,B 0,C 180,E1 3008.294,E2 3008.294} C_VEL
LIN {X 0,Y 714.373,Z 601.31,A -85,B 0,C 180,E1 3013.866,E2 3013.866} C_VEL
LIN {X 0,Y 714.106,Z 601.31,A -85,B 0,C 180,E1 3018.883,E2 3018.883} C_VEL
LIN {X 0,Y 714.148,Z 601.31,A -85,B 0,C 180,E1 3023.725,E2 3023.725} C_VEL
LIN {X 0,Y 714.243,Z 601.31,A -85,B 0,C 180,E1 3029.403,E2 3029.403} C_VEL
LIN {X 0,Y 714.315,Z 601.31,A -85,B 0,C 180,E1 3034.905,E2 3034.905} C_VEL
LIN {X 0,Y 714.154,Z 601.31,A -85,B 0,C 180,E1 3038.984,E2 3038.984} C_VEL
LIN {X 0,Y 714.294,Z 601.31,A -85,B 0,C 180,E1 3042.014,E2 3042.014} C_VEL
LIN {X 0,Y 717.034,Z 614.715,A -85,B 0,C 180,E1 3042.234,E2 3042.234} C_VEL
LIN {X 0,Y 716.904,Z 691.419,A -85,B 0,C 180,E1 3043.111,E2 3043.111} C_VEL
LIN {X 0,Y 716.596,Z 724.644,A -85,B 0,C 180,E1 3043.972,E2 3043.972} C_VEL
LIN {X 0,Y 716.122,Z 756.344,A -85,B 0,C 180,E1 3045.296,E2 3045.296} C_VEL
LIN {X 0,Y 715.632,Z 784.764,A -85,B 0,C 180,E1 3047.014,E2 3047.014} C_VEL
LIN {X 0,Y 715.21,Z 810.168,A -85,B 0,C 180,E1 3049.167,E2 3049.167} C_VEL
LIN {X 0,Y 714.96,Z 829.503,A -85,B 0,C 180,E1 3051.472,E2 3051.472} C_VEL
LIN {X 0,Y 714.841,Z 843.795,A -85,B 0,C 180,E1 3053.919,E2 3053.919} C_VEL
LIN {X 0,Y 714.772,Z 852.685,A -85,B 0,C 180,E1 3056.356,E2 3056.356} C_VEL
LIN {X 0,Y 714.702,Z 856.957,A -85,B 0,C 180,E1 3058.787,E2 3058.787} C_VEL
LIN {X 0,Y 714.723,Z 856.878,A -85,B 0,C 180,E1 3061.216,E2 3061.216} C_VEL
LIN {X 0,Y 714.793,Z 852.445,A -85,B 0,C 180,E1 3063.647,E2 3063.647} C_VEL
LIN {X 0,Y 714.851,Z 841.81,A -85,B 0,C 180,E1 3066.389,E2 3066.389} C_VEL
LIN {X 0,Y 715.03,Z 825.455,A -85,B 0,C 180,E1 3068.991,E2 3068.991} C_VEL
LIN {X 0,Y 715.033,Z 821.643,A -85,B 0,C 180,E1 3069.475,E2 3069.475} C_VEL
LIN {X 0,Y 711.203,Z 811.996,A -85,B 0,C 180,E1 3070.613,E2 3070.613} C_VEL
LIN {X 0,Y 707.524,Z 801.36,A -85,B 0,C 180,E1 3071.701,E2 3071.701} C_VEL
LIN {X 0,Y 708.053,Z 775.23,A -85,B 0,C 180,E1 3073.692,E2 3073.692} C_VEL
LIN {X 0,Y 708.587,Z 745.382,A -85,B 0,C 180,E1 3075.304,E2 3075.304} C_VEL
LIN {X 0,Y 709.137,Z 712.667,A -85,B 0,C 180,E1 3076.484,E2 3076.484} C_VEL
LIN {X 0,Y 709.428,Z 678.359,A -85,B 0,C 180,E1 3077.196,E2 3077.196} C_VEL
LIN {X 0,Y 708.692,Z 609.677,A -85,B 0,C 180,E1 3077.954,E2 3077.954} C_VEL
LIN {X 0,Y 706.571,Z 601.31,A -85,B 0,C 180,E1 3078.114,E2 3078.114} C_VEL
LIN {X 0,Y 706.301,Z 601.31,A -85,B 0,C 180,E1 3082.72,E2 3082.72} C_VEL
LIN {X 0,Y 706.307,Z 601.31,A -85,B 0,C 180,E1 3086.771,E2 3086.771} C_VEL
LIN {X 0,Y 706.301,Z 601.31,A -85,B 0,C 180,E1 3090.983,E2 3090.983} C_VEL
LIN {X 0,Y 706.268,Z 601.31,A -85,B 0,C 180,E1 3095.395,E2 3095.395} C_VEL
LIN {X 0,Y 706.16,Z 601.31,A -85,B 0,C 180,E1 3100.061,E2 3100.061} C_VEL
LIN {X 0,Y 706.4,Z 601.31,A -85,B 0,C 180,E1 3105.049,E2 3105.049} C_VEL
LIN {X 0,Y 706.194,Z 601.31,A -85,B 0,C 180,E1 3110.559,E2 3110.559} C_VEL
LIN {X 0,Y 706.123,Z 601.31,A -85,B 0,C 180,E1 3116.093,E2 3116.093} C_VEL
LIN {X 0,Y 706.154,Z 601.31,A -85,B 0,C 180,E1 3117.448,E2 3117.448} C_VEL
LIN {X 0,Y 714.592,Z 622.121,A -85,B 0,C 180,E1 3118.128,E2 3118.128} C_VEL
LIN {X 0,Y 714.637,Z 707.78,A -85,B 0,C 180,E1 3119.225,E2 3119.225} C_VEL
LIN {X 0,Y 713.721,Z 749.749,A -85,B 0,C 180,E1 3120.201,E2 3120.201} C_VEL
LIN {X 0,Y 712.545,Z 793.898,A -85,B 0,C 180,E1 3121.753,E2 3121.753} C_VEL
LIN {X 0,Y 711.137,Z 836.684,A -85,B 0,C 180,E1 3123.85,E2 3123.85} C_VEL
LIN {X 0,Y 709.842,Z 875.141,A -85,B 0,C 180,E1 3126.335,E2 3126.335} C_VEL
LIN {X 0,Y 708.743,Z 907.774,A -85,B 0,C 180,E1 3129.02,E2 3129.02} C_VEL
LIN {X 0,Y 708.016,Z 935.701,A -85,B 0,C 180,E1 3131.901,E2 3131.901} C_VEL
LIN {X 0,Y 707.359,Z 961.242,A -85,B 0,C 180,E1 3135.267,E2 3135.267} C_VEL
LIN {X 0,Y 706.979,Z 981.634,A -85,B 0,C 180,E1 3138.882,E2 3138.882} C_VEL
LIN {X 0,Y 706.871,Z 994.244,A -85,B 0,C 180,E1 3141.994,E2 3141.994} C_VEL
LIN {X 0,Y 706.75,Z 1003.827,A -85,B 0,C 180,E1 3145.781,E2 3145.781} C_VEL
LIN {X 0,Y 706.808,Z 1007.17,A -85,B 0,C 180,E1 3148.775,E2 3148.775} C_VEL
LIN {X 0,Y 706.821,Z 1006.217,A -85,B 0,C 180,E1 3152.461,E2 3152.461} C_VEL
LIN {X 0,Y 706.786,Z 999.627,A -85,B 0,C 180,E1 3156.157,E2 3156.157} C_VEL
LIN {X 0,Y 706.891,Z 988.093,A -85,B 0,C 180,E1 3159.662,E2 3159.662} C_VEL
LIN {X 0,Y 707.079,Z 971.512,A -85,B 0,C 180,E1 3163.053,E2 3163.053} C_VEL
LIN {X 0,Y 707.483,Z 949.958,A -85,B 0,C 180,E1 3166.329,E2 3166.329} C_VEL
LIN {X 0,Y 708.212,Z 922.904,A -85,B 0,C 180,E1 3169.508,E2 3169.508} C_VEL
LIN {X 0,Y 709.336,Z 890.181,A -85,B 0,C 180,E1 3172.511,E2 3172.511} C_VEL
LIN {X 0,Y 710.621,Z 851.914,A -85,B 0,C 180,E1 3175.246,E2 3175.246} C_VEL
LIN {X 0,Y 712.054,Z 810.83,A -85,B 0,C 180,E1 3177.487,E2 3177.487} C_VEL
LIN {X 0,Y 713.249,Z 770.808,A -85,B 0,C 180,E1 3179.122,E2 3179.122} C_VEL
LIN {X 0,Y 714.324,Z 728.719,A -85,B 0,C 180,E1 3180.345,E2 3180.345} C_VEL
LIN {X 0,Y 714.829,Z 684.316,A -85,B 0,C 180,E1 3181.134,E2 3181.134} C_VEL
LIN {X 0,Y 714.452,Z 619.848,A -85,B 0,C 180,E1 3181.905,E2 3181.905} C_VEL
LIN {X 0,Y 706.522,Z 601.31,A -85,B 0,C 180,E1 3182.565,E2 3182.565} C_VEL
LIN {X 0,Y 706.217,Z 601.31,A -85,B 0,C 180,E1 3187.467,E2 3187.467} C_VEL
LIN {X 0,Y 706.409,Z 601.31,A -85,B 0,C 180,E1 3193.349,E2 3193.349} C_VEL
LIN {X 0,Y 706.179,Z 601.31,A -85,B 0,C 180,E1 3198.68,E2 3198.68} C_VEL
LIN {X 0,Y 706.153,Z 601.31,A -85,B 0,C 180,E1 3203.08,E2 3203.08} C_VEL
LIN {X 0,Y 706.215,Z 601.31,A -85,B 0,C 180,E1 3207.568,E2 3207.568} C_VEL
LIN {X 0,Y 706.265,Z 601.31,A -85,B 0,C 180,E1 3211.842,E2 3211.842} C_VEL
LIN {X 0,Y 706.399,Z 601.31,A -85,B 0,C 180,E1 3215.953,E2 3215.953} C_VEL
LIN {X 0,Y 706.4,Z 601.31,A -85,B 0,C 180,E1 3221.234,E2 3221.234} C_VEL
LIN {X 0,Y 706.319,Z 601.31,A -85,B 0,C 180,E1 3226.352,E2 3226.352} C_VEL
LIN {X 0,Y 706.411,Z 601.31,A -85,B 0,C 180,E1 3231.365,E2 3231.365} C_VEL
LIN {X 0,Y 706.6,Z 601.31,A -85,B 0,C 180,E1 3236.311,E2 3236.311} C_VEL
LIN {X 0,Y 706.748,Z 601.31,A -85,B 0,C 180,E1 3241.227,E2 3241.227} C_VEL
LIN {X 0,Y 706.477,Z 601.31,A -85,B 0,C 180,E1 3246.153,E2 3246.153} C_VEL
LIN {X 0,Y 706.428,Z 601.31,A -85,B 0,C 180,E1 3251.126,E2 3251.126} C_VEL
LIN {X 0,Y 706.506,Z 601.31,A -85,B 0,C 180,E1 3256.184,E2 3256.184} C_VEL
LIN {X 0,Y 706.42,Z 601.31,A -85,B 0,C 180,E1 3261.379,E2 3261.379} C_VEL
LIN {X 0,Y 706.319,Z 601.31,A -85,B 0,C 180,E1 3265.704,E2 3265.704} C_VEL
LIN {X 0,Y 706.288,Z 601.31,A -85,B 0,C 180,E1 3270.98,E2 3270.98} C_VEL
LIN {X 0,Y 706.255,Z 601.31,A -85,B 0,C 180,E1 3275.388,E2 3275.388} C_VEL
LIN {X 0,Y 706.156,Z 601.31,A -85,B 0,C 180,E1 3280.057,E2 3280.057} C_VEL
LIN {X 0,Y 706.376,Z 601.31,A -85,B 0,C 180,E1 3285.047,E2 3285.047} C_VEL
LIN {X 0,Y 706.223,Z 601.31,A -85,B 0,C 180,E1 3290.551,E2 3290.551} C_VEL
LIN {X 0,Y 706.196,Z 601.31,A -85,B 0,C 180,E1 3296.089,E2 3296.089} C_VEL
LIN {X 0,Y 706.283,Z 601.31,A -85,B 0,C 180,E1 3300.43,E2 3300.43} C_VEL
LIN {X 0,Y 706.558,Z 601.31,A -85,B 0,C 180,E1 3305.388,E2 3305.388} C_VEL
LIN {X 0,Y 711.55,Z 619.629,A -85,B 0,C 180,E1 3305.851,E2 3305.851} C_VEL
LIN {X 0,Y 711.039,Z 661.414,A -85,B 0,C 180,E1 3306.859,E2 3306.859} C_VEL
LIN {X 0,Y 710.207,Z 699.647,A -85,B 0,C 180,E1 3308.301,E2 3308.301} C_VEL
LIN {X 0,Y 709.201,Z 735.965,A -85,B 0,C 180,E1 3310.235,E2 3310.235} C_VEL
LIN {X 0,Y 708.288,Z 768.611,A -85,B 0,C 180,E1 3312.569,E2 3312.569} C_VEL
LIN {X 0,Y 707.597,Z 795.516,A -85,B 0,C 180,E1 3315.107,E2 3315.107} C_VEL
LIN {X 0,Y 707.196,Z 818.286,A -85,B 0,C 180,E1 3317.939,E2 3317.939} C_VEL
LIN {X 0,Y 706.912,Z 835.448,A -85,B 0,C 180,E1 3320.831,E2 3320.831} C_VEL
LIN {X 0,Y 706.783,Z 847.743,A -85,B 0,C 180,E1 3323.843,E2 3323.843} C_VEL
LIN {X 0,Y 706.774,Z 854.029,A -85,B 0,C 180,E1 3326.309,E2 3326.309} C_VEL
LIN {X 0,Y 706.704,Z 857.09,A -85,B 0,C 180,E1 3328.768,E2 3328.768} C_VEL
LIN {X 0,Y 706.789,Z 857.03,A -85,B 0,C 180,E1 3331.225,E2 3331.225} C_VEL
LIN {X 0,Y 706.882,Z 852.632,A -85,B 0,C 180,E1 3334.277,E2 3334.277} C_VEL
LIN {X 0,Y 706.899,Z 843.019,A -85,B 0,C 180,E1 3337.386,E2 3337.386} C_VEL
LIN {X 0,Y 707.056,Z 827.814,A -85,B 0,C 180,E1 3340.492,E2 3340.492} C_VEL
LIN {X 0,Y 707.476,Z 805.833,A -85,B 0,C 180,E1 3343.623,E2 3343.623} C_VEL
LIN {X 0,Y 708.032,Z 780.436,A -85,B 0,C 180,E1 3346.309,E2 3346.309} C_VEL
LIN {X 0,Y 708.807,Z 750.721,A -85,B 0,C 180,E1 3348.699,E2 3348.699} C_VEL
LIN {X 0,Y 709.699,Z 716.52,A -85,B 0,C 180,E1 3350.786,E2 3350.786} C_VEL
LIN {X 0,Y 710.64,Z 679.748,A -85,B 0,C 180,E1 3352.43,E2 3352.43} C_VEL
LIN {X 0,Y 711.409,Z 639.569,A -85,B 0,C 180,E1 3353.643,E2 3353.643} C_VEL
LIN {X 0,Y 710.988,Z 615.009,A -85,B 0,C 180,E1 3354.161,E2 3354.161} C_VEL
LIN {X 0,Y 706.303,Z 601.31,A -85,B 0,C 180,E1 3354.579,E2 3354.579} C_VEL
LIN {X 0,Y 706.271,Z 601.31,A -85,B 0,C 180,E1 3359.563,E2 3359.563} C_VEL
LIN {X 0,Y 706.239,Z 601.31,A -85,B 0,C 180,E1 3363.901,E2 3363.901} C_VEL
LIN {X 0,Y 706.204,Z 601.31,A -85,B 0,C 180,E1 3368.474,E2 3368.474} C_VEL
LIN {X 0,Y 706.418,Z 601.31,A -85,B 0,C 180,E1 3373.339,E2 3373.339} C_VEL
LIN {X 0,Y 706.194,Z 601.31,A -85,B 0,C 180,E1 3378.668,E2 3378.668} C_VEL
LIN {X 0,Y 706.16,Z 601.31,A -85,B 0,C 180,E1 3383.084,E2 3383.084} C_VEL
LIN {X 0,Y 706.236,Z 601.31,A -85,B 0,C 180,E1 3387.573,E2 3387.573} C_VEL
LIN {X 0,Y 706.409,Z 601.31,A -85,B 0,C 180,E1 3393.236,E2 3393.236} C_VEL
LIN {X 0,Y 706.426,Z 601.31,A -85,B 0,C 180,E1 3397.296,E2 3397.296} C_VEL
LIN {X 0,Y 706.339,Z 601.31,A -85,B 0,C 180,E1 3401.802,E2 3401.802} C_VEL
LIN {X 0,Y 709.558,Z 617.757,A -85,B 0,C 180,E1 3402.071,E2 3402.071} C_VEL
LIN {X 0,Y 709.36,Z 691.393,A -85,B 0,C 180,E1 3402.926,E2 3402.926} C_VEL
LIN {X 0,Y 709.002,Z 724.629,A -85,B 0,C 180,E1 3403.795,E2 3403.795} C_VEL
LIN {X 0,Y 708.435,Z 756.33,A -85,B 0,C 180,E1 3405.133,E2 3405.133} C_VEL
LIN {X 0,Y 707.883,Z 784.755,A -85,B 0,C 180,E1 3406.869,E2 3406.869} C_VEL
LIN {X 0,Y 707.392,Z 810.163,A -85,B 0,C 180,E1 3409.045,E2 3409.045} C_VEL
LIN {X 0,Y 707.062,Z 830.584,A -85,B 0,C 180,E1 3411.531,E2 3411.531} C_VEL
LIN {X 0,Y 706.911,Z 845.133,A -85,B 0,C 180,E1 3414.159,E2 3414.159} C_VEL
LIN {X 0,Y 706.858,Z 854.198,A -85,B 0,C 180,E1 3416.93,E2 3416.93} C_VEL
LIN {X 0,Y 706.815,Z 856.956,A -85,B 0,C 180,E1 3418.773,E2 3418.773} C_VEL
LIN {X 0,Y 706.834,Z 856.877,A -85,B 0,C 180,E1 3421.23,E2 3421.23} C_VEL
LIN {X 0,Y 706.924,Z 852.446,A -85,B 0,C 180,E1 3423.688,E2 3423.688} C_VEL
LIN {X 0,Y 706.975,Z 841.813,A -85,B 0,C 180,E1 3426.461,E2 3426.461} C_VEL
LIN {X 0,Y 707.165,Z 825.738,A -85,B 0,C 180,E1 3429.055,E2 3429.055} C_VEL
LIN {X 0,Y 707.478,Z 804.414,A -85,B 0,C 180,E1 3431.425,E2 3431.425} C_VEL
LIN {X 0,Y 707.524,Z 801.36,A -85,B 0,C 180,E1 3431.701,E2 3431.701} C_VEL
LIN {X 0,Y 704.027,Z 789.874,A -85,B 0,C 180,E1 3432.729,E2 3432.729} C_VEL
LIN {X 0,Y 700.299,Z 777.418,A -85,B 0,C 180,E1 3433.701,E2 3433.701} C_VEL
LIN {X 0,Y 700.881,Z 748.007,A -85,B 0,C 180,E1 3435.355,E2 3435.355} C_VEL
LIN {X 0,Y 701.521,Z 715.711,A -85,B 0,C 180,E1 3436.587,E2 3436.587} C_VEL
LIN {X 0,Y 701.911,Z 681.802,A -85,B 0,C 180,E1 3437.345,E2 3437.345} C_VEL
LIN {X 0,Y 701.3,Z 611.137,A -85,B 0,C 180,E1 3438.166,E2 3438.166} C_VEL
LIN {X 0,Y 698.66,Z 601.31,A -85,B 0,C 180,E1 3438.384,E2 3438.384} C_VEL
LIN {X 0,Y 698.412,Z 601.31,A -85,B 0,C 180,E1 3442.983,E2 3442.983} C_VEL
LIN {X 0,Y 698.386,Z 601.31,A -85,B 0,C 180,E1 3447.194,E2 3447.194} C_VEL
LIN {X 0,Y 698.38,Z 601.31,A -85,B 0,C 180,E1 3452.212,E2 3452.212} C_VEL
LIN {X 0,Y 698.411,Z 601.31,A -85,B 0,C 180,E1 3457.399,E2 3457.399} C_VEL
LIN {X 0,Y 698.397,Z 601.31,A -85,B 0,C 180,E1 3462.474,E2 3462.474} C_VEL
LIN {X 0,Y 698.21,Z 601.31,A -85,B 0,C 180,E1 3467.726,E2 3467.726} C_VEL
LIN {X 0,Y 698.251,Z 601.31,A -85,B 0,C 180,E1 3472.588,E2 3472.588} C_VEL
LIN {X 0,Y 698.225,Z 601.31,A -85,B 0,C 180,E1 3477.012,E2 3477.012} C_VEL
LIN {X 0,Y 708.173,Z 625.565,A -85,B 0,C 180,E1 3477.845,E2 3477.845} C_VEL
LIN {X 0,Y 707.831,Z 707.912,A -85,B 0,C 180,E1 3478.899,E2 3478.899} C_VEL
LIN {X 0,Y 706.823,Z 749.577,A -85,B 0,C 180,E1 3479.875,E2 3479.875} C_VEL
LIN {X 0,Y 705.463,Z 794.184,A -85,B 0,C 180,E1 3481.457,E2 3481.457} C_VEL
LIN {X 0,Y 703.889,Z 837.148,A -85,B 0,C 180,E1 3483.586,E2 3483.586} C_VEL
LIN {X 0,Y 702.371,Z 876.317,A -85,B 0,C 180,E1 3486.155,E2 3486.155} C_VEL
LIN {X 0,Y 701.107,Z 909.529,A -85,B 0,C 180,E1 3488.947,E2 3488.947} C_VEL
LIN {X 0,Y 700.16,Z 938.37,A -85,B 0,C 180,E1 3492.015,E2 3492.015} C_VEL
LIN {X 0,Y 699.527,Z 962.271,A -85,B 0,C 180,E1 3495.259,E2 3495.259} C_VEL
LIN {X 0,Y 699.108,Z 983.157,A -85,B 0,C 180,E1 3499.072,E2 3499.072} C_VEL
LIN {X 0,Y 698.882,Z 996.17,A -85,B 0,C 180,E1 3502.529,E2 3502.529} C_VEL
LIN {X 0,Y 698.855,Z 1003.714,A -85,B 0,C 180,E1 3505.674,E2 3505.674} C_VEL
LIN {X 0,Y 698.905,Z 1007.17,A -85,B 0,C 180,E1 3508.761,E2 3508.761} C_VEL
LIN {X 0,Y 698.915,Z 1006.216,A -85,B 0,C 180,E1 3512.488,E2 3512.488} C_VEL
LIN {X 0,Y 698.882,Z 999.627,A -85,B 0,C 180,E1 3516.227,E2 3516.227} C_VEL
LIN {X 0,Y 699.004,Z 988.677,A -85,B 0,C 180,E1 3519.634,E2 3519.634} C_VEL
LIN {X 0,Y 699.228,Z 971.188,A -85,B 0,C 180,E1 3523.261,E2 3523.261} C_VEL
LIN {X 0,Y 699.675,Z 949.957,A -85,B 0,C 180,E1 3526.517,E2 3526.517} C_VEL
LIN {X 0,Y 700.54,Z 922.657,A -85,B 0,C 180,E1 3529.755,E2 3529.755} C_VEL
LIN {X 0,Y 701.78,Z 890.794,A -85,B 0,C 180,E1 3532.716,E2 3532.716} C_VEL
LIN {X 0,Y 703.301,Z 851.914,A -85,B 0,C 180,E1 3535.527,E2 3535.527} C_VEL
LIN {X 0,Y 704.907,Z 810.826,A -85,B 0,C 180,E1 3537.79,E2 3537.79} C_VEL
LIN {X 0,Y 706.268,Z 770.81,A -85,B 0,C 180,E1 3539.438,E2 3539.438} C_VEL
LIN {X 0,Y 707.42,Z 730.671,A -85,B 0,C 180,E1 3540.625,E2 3540.625} C_VEL
LIN {X 0,Y 708.06,Z 685.733,A -85,B 0,C 180,E1 3541.445,E2 3541.445} C_VEL
